KUKA KRL program: f1_Kuka_APT211T03S11.SRC

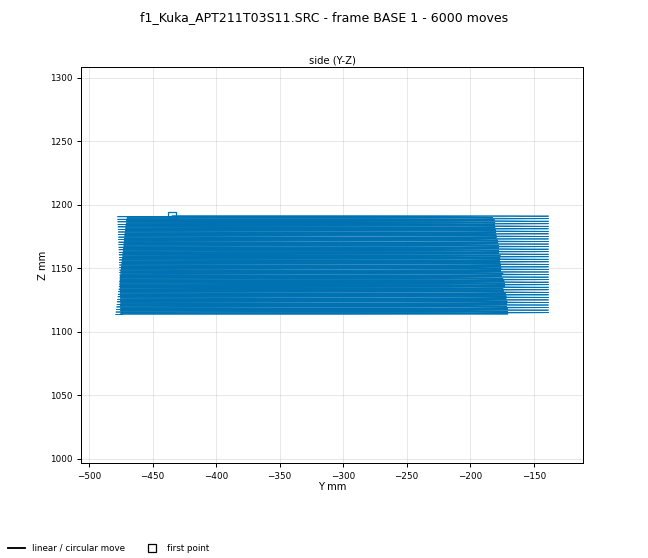
[picture p0: tool path of f1_Kuka_APT211T03S11.SRC in frame BASE 1, 6000 of 6001 moves have a stored position in this frame; points joined in program order, loops and branches not executed]
&ACCESS RVP
&REL 2
&PARAM TEMPLATE = C:\KRC\Roboter\Template\vorgabe
&PARAM EDITMASK = *
DEF f1_Kuka_APT211T03S11()


;FOLD INI;%{PE}%V3.2.0,%MKUKATPBASIS,%CINIT,%VCOMMON,%P
  ;FOLD BAS INI;%{E}%V3.2.0,%MKUKATPBASIS,%CINIT,%VINIT,%P
    GLOBAL INTERRUPT DECL 3 WHEN $STOPMESS==TRUE DO IR_STOPM ( )
    INTERRUPT ON 3
    BAS (#INITMOV,0 )
  ;ENDFOLD (BAS INI)
  ;FOLD USER INI;%{E}%V3.2.0,%MKUKATPUSER,%CINIT,%VINIT,%P
    ;Make your modifications here
  ;ENDFOLD (USER INI)
;ENDFOLD (INI)


;*** Make Null PTP Move
  PTP $pos_act

;*** Auto Load The Correct TOOL Data
  $tool=tool_data[3]

;*** Auto Load The Correct BASE Data
  $base=base_data[1]

  $ADVANCE = 5

;*** Restate Last Velocity
MMPM(30000.0)
SetRPM(6000)
LIN {X -0.088,Y -434.783,Z 1191.509,A 0.000,B 0.000,C 90.000,E1 271.661} C_DIS
LIN {X 0.189,Y -427.658,Z 1191.507,A 0.000,B 0.000,C 90.000,E1 271.318} C_DIS
LIN {X 0.032,Y -420.756,Z 1191.506,A 0.000,B 0.000,C 90.000,E1 271.088} C_DIS
LIN {X -0.167,Y -410.743,Z 1191.504,A 0.000,B 0.000,C 90.000,E1 270.802} C_DIS
LIN {X 0.135,Y -403.684,Z 1191.503,A 0.000,B 0.000,C 90.000,E1 270.573} C_DIS
LIN {X 0.127,Y -392.814,Z 1191.502,A 0.000,B 0.000,C 90.000,E1 270.344} C_DIS
LIN {X 0.051,Y -385.052,Z 1191.501,A 0.000,B 0.000,C 90.000,E1 270.229} C_DIS
LIN {X 0.126,Y -375.484,Z 1191.501,A 0.000,B 0.000,C 90.000,E1 270.115} C_DIS
LIN {X -0.096,Y -368.887,Z 1191.501,A 0.000,B 0.000,C 90.000,E1 270.115} C_DIS
LIN {X -0.083,Y -181.572,Z 1191.500,A 0.000,B 0.000,C 90.000,E1 270.115} C_DIS
LIN {X 0.017,Y -180.908,Z 1191.475,A 0.000,B 0.000,C 90.000,E1 265.527} C_DIS
LIN {X 0.075,Y -180.763,Z 1191.470,A 0.000,B 0.000,C 90.000,E1 264.666} C_DIS
LIN {X -0.034,Y -178.857,Z 1191.442,A 0.000,B 0.000,C 90.000,E1 259.634} C_DIS
LIN {X 0.037,Y -175.900,Z 1191.414,A 0.000,B 0.000,C 90.000,E1 254.519} C_DIS
LIN {X -0.024,Y -174.579,Z 1191.405,A 0.000,B 0.000,C 90.000,E1 252.834} C_DIS
LIN {X 0.011,Y -171.562,Z 1191.381,A 0.000,B 0.000,C 90.000,E1 248.539} C_DIS
LIN {X -0.006,Y -167.786,Z 1191.357,A 0.000,B 0.000,C 90.000,E1 244.229} C_DIS
LIN {X 0.008,Y -166.499,Z 1191.347,A 0.000,B 0.000,C 90.000,E1 242.487} C_DIS
LIN {X 0.004,Y -163.209,Z 1191.328,A 0.000,B 0.000,C 90.000,E1 238.997} C_DIS
LIN {X -0.032,Y -161.174,Z 1191.313,A 0.000,B 0.000,C 90.000,E1 236.373} C_DIS
LIN {X 0.093,Y -157.187,Z 1191.289,A 0.000,B 0.000,C 90.000,E1 231.904} C_DIS
LIN {X 0.015,Y -155.917,Z 1191.279,A 0.000,B 0.000,C 90.000,E1 230.150} C_DIS
LIN {X 0.071,Y -152.169,Z 1191.254,A 0.000,B 0.000,C 90.000,E1 225.648} C_DIS
LIN {X -0.020,Y -150.416,Z 1191.239,A 0.000,B 0.000,C 90.000,E1 222.975} C_DIS
LIN {X -0.094,Y -147.145,Z 1191.214,A 0.000,B 0.000,C 90.000,E1 218.463} C_DIS
LIN {X 0.019,Y -145.703,Z 1191.198,A 0.000,B 0.000,C 90.000,E1 215.678} C_DIS
LIN {X 0.027,Y -143.087,Z 1191.173,A 0.000,B 0.000,C 90.000,E1 211.082} C_DIS
LIN {X 0.032,Y -141.703,Z 1191.152,A 0.000,B 0.000,C 90.000,E1 207.385} C_DIS
LIN {X -0.046,Y -139.468,Z 1191.116,A 0.000,B 0.000,C 90.000,E1 200.918} C_DIS
LIN {X 0.008,Y -139.201,Z 1191.106,A 0.000,B 0.000,C 90.000,E1 199.033} C_DIS
LIN {X 0.071,Y -138.327,Z 1191.054,A 0.000,B 0.000,C 90.000,E1 189.670} C_DIS
LIN {X -0.062,Y -139.443,Z 1191.007,A 0.000,B 0.000,C 90.000,E1 181.318} C_DIS
LIN {X 0.017,Y -140.980,Z 1190.976,A 0.000,B 0.000,C 90.000,E1 175.698} C_DIS
LIN {X -0.033,Y -142.736,Z 1190.956,A 0.000,B 0.000,C 90.000,E1 172.008} C_DIS
LIN {X 0.066,Y -145.126,Z 1190.930,A 0.000,B 0.000,C 90.000,E1 167.353} C_DIS
LIN {X 0.059,Y -147.749,Z 1190.910,A 0.000,B 0.000,C 90.000,E1 163.685} C_DIS
LIN {X -0.001,Y -150.418,Z 1190.889,A 0.000,B 0.000,C 90.000,E1 160.061} C_DIS
LIN {X 0.014,Y -153.858,Z 1190.869,A 0.000,B 0.000,C 90.000,E1 156.433} C_DIS
LIN {X -0.069,Y -157.269,Z 1190.849,A 0.000,B 0.000,C 90.000,E1 152.871} C_DIS
LIN {X 0.008,Y -161.446,Z 1190.829,A 0.000,B 0.000,C 90.000,E1 149.282} C_DIS
LIN {X 0.016,Y -165.646,Z 1190.810,A 0.000,B 0.000,C 90.000,E1 145.754} C_DIS
LIN {X -0.002,Y -170.580,Z 1190.790,A 0.000,B 0.000,C 90.000,E1 142.271} C_DIS
LIN {X -0.095,Y -175.457,Z 1190.771,A 0.000,B 0.000,C 90.000,E1 138.852} C_DIS
LIN {X 0.020,Y -181.080,Z 1190.752,A 0.000,B 0.000,C 90.000,E1 135.405} C_DIS
LIN {X 0.010,Y -186.520,Z 1190.734,A 0.000,B 0.000,C 90.000,E1 132.043} C_DIS
LIN {X -0.048,Y -191.139,Z 1190.720,A 0.000,B 0.000,C 90.000,E1 129.564} C_DIS
LIN {X 0.030,Y -196.938,Z 1190.701,A 0.000,B 0.000,C 90.000,E1 126.251} C_DIS
LIN {X -0.015,Y -201.163,Z 1190.690,A 0.000,B 0.000,C 90.000,E1 124.119} C_DIS
LIN {X 0.133,Y -201.443,Z 1190.689,A 0.000,B 0.000,C 90.000,E1 123.913} C_DIS
LIN {X 0.171,Y -311.509,Z 1190.689,A 0.000,B 0.000,C 90.000,E1 123.913} C_DIS
LIN {X -0.067,Y -315.813,Z 1190.688,A 0.000,B 0.000,C 90.000,E1 123.833} C_DIS
LIN {X 0.069,Y -318.680,Z 1190.687,A 0.000,B 0.000,C 90.000,E1 123.627} C_DIS
LIN {X 0.063,Y -322.419,Z 1190.685,A 0.000,B 0.000,C 90.000,E1 123.245} C_DIS
LIN {X 0.082,Y -325.877,Z 1190.682,A 0.000,B 0.000,C 90.000,E1 122.673} C_DIS
LIN {X -0.013,Y -328.378,Z 1190.678,A 0.000,B 0.000,C 90.000,E1 122.054} C_DIS
LIN {X 0.171,Y -339.358,Z 1190.662,A 0.000,B 0.000,C 90.000,E1 119.205} C_DIS
LIN {X -0.121,Y -351.728,Z 1190.647,A 0.000,B 0.000,C 90.000,E1 116.488} C_DIS
LIN {X -0.053,Y -365.589,Z 1190.632,A 0.000,B 0.000,C 90.000,E1 113.770} C_DIS
LIN {X 0.003,Y -379.265,Z 1190.619,A 0.000,B 0.000,C 90.000,E1 111.408} C_DIS
LIN {X 0.128,Y -394.313,Z 1190.606,A 0.000,B 0.000,C 90.000,E1 109.087} C_DIS
LIN {X -0.003,Y -410.841,Z 1190.594,A 0.000,B 0.000,C 90.000,E1 106.858} C_DIS
LIN {X 0.038,Y -428.965,Z 1190.582,A 0.000,B 0.000,C 90.000,E1 104.662} C_DIS
LIN {X 0.172,Y -448.597,Z 1190.570,A 0.000,B 0.000,C 90.000,E1 102.535} C_DIS
LIN {X 0.088,Y -471.379,Z 1190.558,A 0.000,B 0.000,C 90.000,E1 100.366} C_DIS
LIN {X -0.023,Y -473.312,Z 1190.556,A 0.000,B 0.000,C 90.000,E1 100.141} C_DIS
LIN {X -0.052,Y -474.780,Z 1190.555,A 0.000,B 0.000,C 90.000,E1 99.905} C_DIS
LIN {X 0.143,Y -476.796,Z 1190.552,A 0.000,B 0.000,C 90.000,E1 99.378} C_DIS
LIN {X -0.202,Y -477.678,Z 1190.549,A 0.000,B 0.000,C 90.000,E1 98.916} C_DIS
LIN {X -0.062,Y -477.576,Z 1190.547,A 0.000,B 0.000,C 90.000,E1 98.398} C_DIS
LIN {X 0.151,Y -476.484,Z 1190.544,A 0.000,B 0.000,C 90.000,E1 97.871} C_DIS
LIN {X -0.044,Y -475.517,Z 1190.542,A 0.000,B 0.000,C 90.000,E1 97.644} C_DIS
LIN {X -0.176,Y -474.208,Z 1190.541,A 0.000,B 0.000,C 90.000,E1 97.409} C_DIS
LIN {X -0.051,Y -461.532,Z 1190.531,A 0.000,B 0.000,C 90.000,E1 95.625} C_DIS
LIN {X -0.170,Y -448.957,Z 1190.521,A 0.000,B 0.000,C 90.000,E1 93.841} C_DIS
LIN {X 0.191,Y -433.692,Z 1190.508,A 0.000,B 0.000,C 90.000,E1 91.432} C_DIS
LIN {X 0.019,Y -421.108,Z 1190.496,A 0.000,B 0.000,C 90.000,E1 89.312} C_DIS
LIN {X -0.088,Y -410.843,Z 1190.486,A 0.000,B 0.000,C 90.000,E1 87.421} C_DIS
LIN {X 0.017,Y -400.562,Z 1190.475,A 0.000,B 0.000,C 90.000,E1 85.469} C_DIS
LIN {X -0.061,Y -390.360,Z 1190.464,A 0.000,B 0.000,C 90.000,E1 83.514} C_DIS
LIN {X 0.119,Y -380.156,Z 1190.453,A 0.000,B 0.000,C 90.000,E1 81.489} C_DIS
LIN {X 0.144,Y -371.127,Z 1190.443,A 0.000,B 0.000,C 90.000,E1 79.746} C_DIS
LIN {X 0.074,Y -361.815,Z 1190.433,A 0.000,B 0.000,C 90.000,E1 77.993} C_DIS
LIN {X -0.083,Y -352.243,Z 1190.423,A 0.000,B 0.000,C 90.000,E1 76.228} C_DIS
LIN {X -0.072,Y -340.984,Z 1190.412,A 0.000,B 0.000,C 90.000,E1 74.102} C_DIS
LIN {X -0.123,Y -329.798,Z 1190.400,A 0.000,B 0.000,C 90.000,E1 71.945} C_DIS
LIN {X -0.013,Y -315.928,Z 1190.384,A 0.000,B 0.000,C 90.000,E1 69.082} C_DIS
LIN {X 0.125,Y -300.034,Z 1190.364,A 0.000,B 0.000,C 90.000,E1 65.485} C_DIS
LIN {X 0.133,Y -287.965,Z 1190.347,A 0.000,B 0.000,C 90.000,E1 62.487} C_DIS
LIN {X -0.085,Y -275.372,Z 1190.328,A 0.000,B 0.000,C 90.000,E1 59.125} C_DIS
LIN {X 0.118,Y -263.526,Z 1190.309,A 0.000,B 0.000,C 90.000,E1 55.595} C_DIS
LIN {X 0.082,Y -253.445,Z 1190.291,A 0.000,B 0.000,C 90.000,E1 52.396} C_DIS
LIN {X 0.059,Y -243.968,Z 1190.273,A 0.000,B 0.000,C 90.000,E1 49.138} C_DIS
LIN {X -0.126,Y -234.043,Z 1190.253,A 0.000,B 0.000,C 90.000,E1 45.486} C_DIS
LIN {X 0.035,Y -224.894,Z 1190.232,A 0.000,B 0.000,C 90.000,E1 41.676} C_DIS
LIN {X -0.024,Y -218.244,Z 1190.215,A 0.000,B 0.000,C 90.000,E1 38.624} C_DIS
LIN {X -0.056,Y -210.782,Z 1190.193,A 0.000,B 0.000,C 90.000,E1 34.739} C_DIS
LIN {X -0.101,Y -204.190,Z 1190.171,A 0.000,B 0.000,C 90.000,E1 30.797} C_DIS
LIN {X 0.043,Y -198.271,Z 1190.149,A 0.000,B 0.000,C 90.000,E1 26.744} C_DIS
LIN {X -0.001,Y -193.148,Z 1190.126,A 0.000,B 0.000,C 90.000,E1 22.695} C_DIS
LIN {X -0.037,Y -188.788,Z 1190.103,A 0.000,B 0.000,C 90.000,E1 18.598} C_DIS
LIN {X 0.048,Y -185.390,Z 1190.080,A 0.000,B 0.000,C 90.000,E1 14.426} C_DIS
LIN {X 0.061,Y -182.321,Z 1190.048,A 0.000,B 0.000,C 90.000,E1 8.568} C_DIS
LIN {X 0.047,Y -183.292,Z 1189.965,A 0.000,B 0.000,C 90.000,E1 353.628} C_DIS
LIN {X -0.041,Y -186.535,Z 1189.937,A 0.000,B 0.000,C 90.000,E1 348.634} C_DIS
LIN {X 0.062,Y -190.300,Z 1189.914,A 0.000,B 0.000,C 90.000,E1 344.448} C_DIS
LIN {X -0.067,Y -194.984,Z 1189.891,A 0.000,B 0.000,C 90.000,E1 340.369} C_DIS
LIN {X -0.018,Y -200.311,Z 1189.868,A 0.000,B 0.000,C 90.000,E1 336.282} C_DIS
LIN {X 0.077,Y -206.276,Z 1189.846,A 0.000,B 0.000,C 90.000,E1 332.231} C_DIS
LIN {X 0.003,Y -212.819,Z 1189.824,A 0.000,B 0.000,C 90.000,E1 328.280} C_DIS
LIN {X 0.040,Y -219.997,Z 1189.802,A 0.000,B 0.000,C 90.000,E1 324.356} C_DIS
LIN {X 0.105,Y -226.235,Z 1189.785,A 0.000,B 0.000,C 90.000,E1 321.251} C_DIS
LIN {X -0.055,Y -233.325,Z 1189.768,A 0.000,B 0.000,C 90.000,E1 318.243} C_DIS
LIN {X 0.088,Y -242.603,Z 1189.749,A 0.000,B 0.000,C 90.000,E1 314.838} C_DIS
LIN {X 0.016,Y -253.506,Z 1189.731,A 0.000,B 0.000,C 90.000,E1 311.553} C_DIS
LIN {X -0.049,Y -265.573,Z 1189.713,A 0.000,B 0.000,C 90.000,E1 308.338} C_DIS
LIN {X -0.082,Y -275.913,Z 1189.699,A 0.000,B 0.000,C 90.000,E1 305.884} C_DIS
LIN {X 0.028,Y -287.499,Z 1189.686,A 0.000,B 0.000,C 90.000,E1 303.452} C_DIS
LIN {X 0.087,Y -298.373,Z 1189.675,A 0.000,B 0.000,C 90.000,E1 301.416} C_DIS
LIN {X -0.029,Y -312.380,Z 1189.662,A 0.000,B 0.000,C 90.000,E1 299.127} C_DIS
LIN {X 0.042,Y -325.764,Z 1189.651,A 0.000,B 0.000,C 90.000,E1 297.180} C_DIS
LIN {X 0.033,Y -333.126,Z 1189.646,A 0.000,B 0.000,C 90.000,E1 296.232} C_DIS
LIN {X -0.148,Y -354.255,Z 1189.632,A 0.000,B 0.000,C 90.000,E1 293.823} C_DIS
LIN {X 0.035,Y -378.498,Z 1189.618,A 0.000,B 0.000,C 90.000,E1 291.280} C_DIS
LIN {X -0.113,Y -394.625,Z 1189.610,A 0.000,B 0.000,C 90.000,E1 289.758} C_DIS
LIN {X -0.054,Y -407.817,Z 1189.603,A 0.000,B 0.000,C 90.000,E1 288.471} C_DIS
LIN {X -0.106,Y -417.892,Z 1189.597,A 0.000,B 0.000,C 90.000,E1 287.457} C_DIS
LIN {X 0.013,Y -427.679,Z 1189.591,A 0.000,B 0.000,C 90.000,E1 286.386} C_DIS
LIN {X -0.205,Y -434.725,Z 1189.587,A 0.000,B 0.000,C 90.000,E1 285.607} C_DIS
LIN {X 0.060,Y -441.189,Z 1189.582,A 0.000,B 0.000,C 90.000,E1 284.773} C_DIS
LIN {X -0.160,Y -446.904,Z 1189.578,A 0.000,B 0.000,C 90.000,E1 284.008} C_DIS
LIN {X 0.220,Y -451.991,Z 1189.573,A 0.000,B 0.000,C 90.000,E1 283.175} C_DIS
LIN {X 0.095,Y -456.430,Z 1189.569,A 0.000,B 0.000,C 90.000,E1 282.411} C_DIS
LIN {X -0.083,Y -460.057,Z 1189.565,A 0.000,B 0.000,C 90.000,E1 281.658} C_DIS
LIN {X -0.138,Y -463.096,Z 1189.560,A 0.000,B 0.000,C 90.000,E1 280.894} C_DIS
LIN {X -0.015,Y -464.741,Z 1189.558,A 0.000,B 0.000,C 90.000,E1 280.366} C_DIS
LIN {X 0.181,Y -467.347,Z 1189.552,A 0.000,B 0.000,C 90.000,E1 279.321} C_DIS
LIN {X -0.207,Y -468.452,Z 1189.549,A 0.000,B 0.000,C 90.000,E1 278.859} C_DIS
LIN {X -0.123,Y -469.349,Z 1189.546,A 0.000,B 0.000,C 90.000,E1 278.341} C_DIS
LIN {X 0.035,Y -470.033,Z 1189.543,A 0.000,B 0.000,C 90.000,E1 277.814} C_DIS
LIN {X 0.132,Y -470.374,Z 1189.541,A 0.000,B 0.000,C 90.000,E1 277.296} C_DIS
LIN {X 0.234,Y -470.270,Z 1189.538,A 0.000,B 0.000,C 90.000,E1 276.777} C_DIS
LIN {X -0.128,Y -469.820,Z 1189.535,A 0.000,B 0.000,C 90.000,E1 276.315} C_DIS
LIN {X -0.025,Y -468.861,Z 1189.532,A 0.000,B 0.000,C 90.000,E1 275.796} C_DIS
LIN {X 0.075,Y -467.463,Z 1189.529,A 0.000,B 0.000,C 90.000,E1 275.277} C_DIS
LIN {X 0.167,Y -465.601,Z 1189.527,A 0.000,B 0.000,C 90.000,E1 274.759} C_DIS
LIN {X 0.214,Y -463.174,Z 1189.524,A 0.000,B 0.000,C 90.000,E1 274.245} C_DIS
LIN {X -0.181,Y -460.133,Z 1189.521,A 0.000,B 0.000,C 90.000,E1 273.784} C_DIS
LIN {X 0.058,Y -458.329,Z 1189.520,A 0.000,B 0.000,C 90.000,E1 273.498} C_DIS
LIN {X 0.094,Y -453.949,Z 1189.517,A 0.000,B 0.000,C 90.000,E1 272.980} C_DIS
LIN {X -0.130,Y -451.317,Z 1189.515,A 0.000,B 0.000,C 90.000,E1 272.751} C_DIS
LIN {X 0.173,Y -448.439,Z 1189.514,A 0.000,B 0.000,C 90.000,E1 272.465} C_DIS
LIN {X 0.188,Y -442.175,Z 1189.511,A 0.000,B 0.000,C 90.000,E1 272.007} C_DIS
LIN {X -0.055,Y -435.315,Z 1189.509,A 0.000,B 0.000,C 90.000,E1 271.661} C_DIS
LIN {X 0.207,Y -428.243,Z 1189.507,A 0.000,B 0.000,C 90.000,E1 271.318} C_DIS
LIN {X 0.011,Y -421.326,Z 1189.506,A 0.000,B 0.000,C 90.000,E1 271.088} C_DIS
LIN {X 0.195,Y -411.152,Z 1189.504,A 0.000,B 0.000,C 90.000,E1 270.745} C_DIS
LIN {X 0.107,Y -404.249,Z 1189.503,A 0.000,B 0.000,C 90.000,E1 270.573} C_DIS
LIN {X 0.099,Y -393.448,Z 1189.502,A 0.000,B 0.000,C 90.000,E1 270.344} C_DIS
LIN {X 0.008,Y -385.768,Z 1189.501,A 0.000,B 0.000,C 90.000,E1 270.229} C_DIS
LIN {X 0.067,Y -376.435,Z 1189.501,A 0.000,B 0.000,C 90.000,E1 270.115} C_DIS
LIN {X 0.134,Y -365.555,Z 1189.500,A 0.000,B 0.000,C 90.000,E1 270.057} C_DIS
LIN {X 0.046,Y -181.570,Z 1189.500,A 0.000,B 0.000,C 90.000,E1 270.057} C_DIS
LIN {X 0.067,Y -180.855,Z 1189.472,A 0.000,B 0.000,C 90.000,E1 264.951} C_DIS
LIN {X -0.058,Y -178.967,Z 1189.444,A 0.000,B 0.000,C 90.000,E1 259.926} C_DIS
LIN {X -0.047,Y -177.920,Z 1189.435,A 0.000,B 0.000,C 90.000,E1 258.229} C_DIS
LIN {X -0.032,Y -175.556,Z 1189.411,A 0.000,B 0.000,C 90.000,E1 253.976} C_DIS
LIN {X -0.026,Y -172.287,Z 1189.387,A 0.000,B 0.000,C 90.000,E1 249.699} C_DIS
LIN {X -0.048,Y -171.765,Z 1189.382,A 0.000,B 0.000,C 90.000,E1 248.847} C_DIS
LIN {X 0.030,Y -167.366,Z 1189.354,A 0.000,B 0.000,C 90.000,E1 243.640} C_DIS
LIN {X -0.036,Y -166.756,Z 1189.349,A 0.000,B 0.000,C 90.000,E1 242.794} C_DIS
LIN {X 0.024,Y -162.735,Z 1189.325,A 0.000,B 0.000,C 90.000,E1 238.408} C_DIS
LIN {X 0.085,Y -161.426,Z 1189.315,A 0.000,B 0.000,C 90.000,E1 236.628} C_DIS
LIN {X -0.095,Y -157.419,Z 1189.290,A 0.000,B 0.000,C 90.000,E1 232.271} C_DIS
LIN {X 0.059,Y -155.422,Z 1189.275,A 0.000,B 0.000,C 90.000,E1 229.542} C_DIS
LIN {X -0.010,Y -151.747,Z 1189.250,A 0.000,B 0.000,C 90.000,E1 225.081} C_DIS
LIN {X 0.000,Y -149.946,Z 1189.235,A 0.000,B 0.000,C 90.000,E1 222.366} C_DIS
LIN {X 0.028,Y -146.791,Z 1189.210,A 0.000,B 0.000,C 90.000,E1 217.810} C_DIS
LIN {X -0.071,Y -145.365,Z 1189.195,A 0.000,B 0.000,C 90.000,E1 215.105} C_DIS
LIN {X 0.045,Y -142.431,Z 1189.164,A 0.000,B 0.000,C 90.000,E1 209.539} C_DIS
LIN {X -0.031,Y -141.421,Z 1189.149,A 0.000,B 0.000,C 90.000,E1 206.796} C_DIS
LIN {X -0.049,Y -139.362,Z 1189.113,A 0.000,B 0.000,C 90.000,E1 200.301} C_DIS
LIN {X 0.069,Y -138.805,Z 1189.097,A 0.000,B 0.000,C 90.000,E1 197.457} C_DIS
LIN {X -0.012,Y -138.350,Z 1189.056,A 0.000,B 0.000,C 90.000,E1 190.018} C_DIS
LIN {X -0.036,Y -139.544,Z 1189.004,A 0.000,B 0.000,C 90.000,E1 180.688} C_DIS
LIN {X 0.056,Y -141.245,Z 1188.973,A 0.000,B 0.000,C 90.000,E1 175.065} C_DIS
LIN {X 0.015,Y -142.614,Z 1188.957,A 0.000,B 0.000,C 90.000,E1 172.299} C_DIS
LIN {X -0.033,Y -144.930,Z 1188.932,A 0.000,B 0.000,C 90.000,E1 167.701} C_DIS
LIN {X -0.040,Y -147.559,Z 1188.911,A 0.000,B 0.000,C 90.000,E1 164.031} C_DIS
LIN {X -0.009,Y -150.165,Z 1188.891,A 0.000,B 0.000,C 90.000,E1 160.369} C_DIS
LIN {X 0.000,Y -153.538,Z 1188.871,A 0.000,B 0.000,C 90.000,E1 156.741} C_DIS
LIN {X 0.052,Y -156.956,Z 1188.851,A 0.000,B 0.000,C 90.000,E1 153.127} C_DIS
LIN {X -0.012,Y -161.062,Z 1188.831,A 0.000,B 0.000,C 90.000,E1 149.587} C_DIS
LIN {X 0.072,Y -163.170,Z 1188.821,A 0.000,B 0.000,C 90.000,E1 147.788} C_DIS
LIN {X -0.056,Y -167.590,Z 1188.802,A 0.000,B 0.000,C 90.000,E1 144.322} C_DIS
LIN {X -0.011,Y -171.419,Z 1188.787,A 0.000,B 0.000,C 90.000,E1 141.698} C_DIS
LIN {X 0.027,Y -176.336,Z 1188.768,A 0.000,B 0.000,C 90.000,E1 138.243} C_DIS
LIN {X -0.105,Y -180.626,Z 1188.754,A 0.000,B 0.000,C 90.000,E1 135.729} C_DIS
LIN {X 0.010,Y -186.027,Z 1188.735,A 0.000,B 0.000,C 90.000,E1 132.324} C_DIS
LIN {X 0.072,Y -190.663,Z 1188.721,A 0.000,B 0.000,C 90.000,E1 129.806} C_DIS
LIN {X 0.106,Y -196.414,Z 1188.703,A 0.000,B 0.000,C 90.000,E1 126.503} C_DIS
LIN {X -0.033,Y -201.388,Z 1188.689,A 0.000,B 0.000,C 90.000,E1 123.992} C_DIS
LIN {X -0.102,Y -311.074,Z 1188.689,A 0.000,B 0.000,C 90.000,E1 123.992} C_DIS
LIN {X -0.153,Y -312.007,Z 1188.689,A 0.000,B 0.000,C 90.000,E1 123.992} C_DIS
LIN {X 0.048,Y -316.708,Z 1188.688,A 0.000,B 0.000,C 90.000,E1 123.785} C_DIS
LIN {X -0.013,Y -319.086,Z 1188.687,A 0.000,B 0.000,C 90.000,E1 123.627} C_DIS
LIN {X -0.047,Y -322.298,Z 1188.685,A 0.000,B 0.000,C 90.000,E1 123.293} C_DIS
LIN {X -0.078,Y -324.275,Z 1188.683,A 0.000,B 0.000,C 90.000,E1 123.007} C_DIS
LIN {X -0.012,Y -325.822,Z 1188.682,A 0.000,B 0.000,C 90.000,E1 122.704} C_DIS
LIN {X -0.093,Y -328.297,Z 1188.678,A 0.000,B 0.000,C 90.000,E1 122.084} C_DIS
LIN {X -0.195,Y -339.269,Z 1188.662,A 0.000,B 0.000,C 90.000,E1 119.283} C_DIS
LIN {X -0.024,Y -351.630,Z 1188.647,A 0.000,B 0.000,C 90.000,E1 116.488} C_DIS
LIN {X 0.045,Y -365.482,Z 1188.632,A 0.000,B 0.000,C 90.000,E1 113.770} C_DIS
LIN {X 0.101,Y -379.149,Z 1188.619,A 0.000,B 0.000,C 90.000,E1 111.408} C_DIS
LIN {X -0.145,Y -394.188,Z 1188.606,A 0.000,B 0.000,C 90.000,E1 109.141} C_DIS
LIN {X 0.098,Y -410.706,Z 1188.594,A 0.000,B 0.000,C 90.000,E1 106.858} C_DIS
LIN {X 0.139,Y -428.819,Z 1188.582,A 0.000,B 0.000,C 90.000,E1 104.662} C_DIS
LIN {X -0.166,Y -448.444,Z 1188.570,A 0.000,B 0.000,C 90.000,E1 102.591} C_DIS
LIN {X 0.182,Y -471.233,Z 1188.558,A 0.000,B 0.000,C 90.000,E1 100.366} C_DIS
LIN {X 0.075,Y -473.176,Z 1188.556,A 0.000,B 0.000,C 90.000,E1 100.141} C_DIS
LIN {X 0.052,Y -474.653,Z 1188.555,A 0.000,B 0.000,C 90.000,E1 99.905} C_DIS
LIN {X -0.085,Y -475.831,Z 1188.554,A 0.000,B 0.000,C 90.000,E1 99.670} C_DIS
LIN {X 0.247,Y -476.688,Z 1188.552,A 0.000,B 0.000,C 90.000,E1 99.378} C_DIS
LIN {X -0.093,Y -477.583,Z 1188.549,A 0.000,B 0.000,C 90.000,E1 98.916} C_DIS
LIN {X 0.047,Y -477.498,Z 1188.547,A 0.000,B 0.000,C 90.000,E1 98.398} C_DIS
LIN {X 0.259,Y -476.423,Z 1188.544,A 0.000,B 0.000,C 90.000,E1 97.871} C_DIS
LIN {X 0.063,Y -475.465,Z 1188.542,A 0.000,B 0.000,C 90.000,E1 97.644} C_DIS
LIN {X -0.068,Y -474.169,Z 1188.541,A 0.000,B 0.000,C 90.000,E1 97.409} C_DIS
LIN {X 0.053,Y -461.526,Z 1188.531,A 0.000,B 0.000,C 90.000,E1 95.625} C_DIS
LIN {X -0.069,Y -448.940,Z 1188.521,A 0.000,B 0.000,C 90.000,E1 93.841} C_DIS
LIN {X 0.015,Y -432.023,Z 1188.507,A 0.000,B 0.000,C 90.000,E1 91.203} C_DIS
LIN {X -0.190,Y -419.594,Z 1188.495,A 0.000,B 0.000,C 90.000,E1 89.083} C_DIS
LIN {X 0.081,Y -409.356,Z 1188.484,A 0.000,B 0.000,C 90.000,E1 87.135} C_DIS
LIN {X -0.175,Y -397.580,Z 1188.472,A 0.000,B 0.000,C 90.000,E1 84.951} C_DIS
LIN {X 0.116,Y -385.933,Z 1188.459,A 0.000,B 0.000,C 90.000,E1 82.648} C_DIS
LIN {X -0.188,Y -377.121,Z 1188.450,A 0.000,B 0.000,C 90.000,E1 80.971} C_DIS
LIN {X -0.147,Y -367.992,Z 1188.440,A 0.000,B 0.000,C 90.000,E1 79.218} C_DIS
LIN {X 0.086,Y -358.579,Z 1188.430,A 0.000,B 0.000,C 90.000,E1 77.409} C_DIS
LIN {X -0.131,Y -348.939,Z 1188.420,A 0.000,B 0.000,C 90.000,E1 75.644} C_DIS
LIN {X -0.102,Y -337.694,Z 1188.408,A 0.000,B 0.000,C 90.000,E1 73.504} C_DIS
LIN {X 0.157,Y -325.032,Z 1188.394,A 0.000,B 0.000,C 90.000,E1 70.967} C_DIS
LIN {X 0.050,Y -309.920,Z 1188.377,A 0.000,B 0.000,C 90.000,E1 67.794} C_DIS
LIN {X -0.043,Y -294.519,Z 1188.357,A 0.000,B 0.000,C 90.000,E1 64.204} C_DIS
LIN {X -0.078,Y -281.468,Z 1188.338,A 0.000,B 0.000,C 90.000,E1 60.845} C_DIS
LIN {X -0.042,Y -270.440,Z 1188.321,A 0.000,B 0.000,C 90.000,E1 57.740} C_DIS
LIN {X 0.022,Y -259.981,Z 1188.303,A 0.000,B 0.000,C 90.000,E1 54.562} C_DIS
LIN {X 0.039,Y -250.047,Z 1188.285,A 0.000,B 0.000,C 90.000,E1 51.331} C_DIS
LIN {X 0.086,Y -241.753,Z 1188.269,A 0.000,B 0.000,C 90.000,E1 48.405} C_DIS
LIN {X -0.017,Y -231.953,Z 1188.248,A 0.000,B 0.000,C 90.000,E1 44.717} C_DIS
LIN {X 0.079,Y -223.002,Z 1188.227,A 0.000,B 0.000,C 90.000,E1 40.906} C_DIS
LIN {X -0.024,Y -214.998,Z 1188.206,A 0.000,B 0.000,C 90.000,E1 37.076} C_DIS
LIN {X -0.059,Y -207.868,Z 1188.184,A 0.000,B 0.000,C 90.000,E1 33.166} C_DIS
LIN {X 0.052,Y -201.531,Z 1188.162,A 0.000,B 0.000,C 90.000,E1 29.155} C_DIS
LIN {X -0.070,Y -195.841,Z 1188.140,A 0.000,B 0.000,C 90.000,E1 25.155} C_DIS
LIN {X 0.019,Y -191.047,Z 1188.117,A 0.000,B 0.000,C 90.000,E1 21.046} C_DIS
LIN {X 0.037,Y -187.008,Z 1188.094,A 0.000,B 0.000,C 90.000,E1 16.913} C_DIS
LIN {X -0.079,Y -183.534,Z 1188.066,A 0.000,B 0.000,C 90.000,E1 11.951} C_DIS
LIN {X -0.038,Y -181.032,Z 1188.029,A 0.000,B 0.000,C 90.000,E1 5.220} C_DIS
LIN {X -0.034,Y -182.540,Z 1187.969,A 0.000,B 0.000,C 90.000,E1 354.489} C_DIS
LIN {X -0.021,Y -185.557,Z 1187.941,A 0.000,B 0.000,C 90.000,E1 349.454} C_DIS
LIN {X 0.005,Y -189.126,Z 1187.918,A 0.000,B 0.000,C 90.000,E1 345.283} C_DIS
LIN {X 0.025,Y -193.650,Z 1187.895,A 0.000,B 0.000,C 90.000,E1 341.148} C_DIS
LIN {X 0.071,Y -198.868,Z 1187.873,A 0.000,B 0.000,C 90.000,E1 337.050} C_DIS
LIN {X -0.064,Y -204.695,Z 1187.850,A 0.000,B 0.000,C 90.000,E1 333.050} C_DIS
LIN {X -0.105,Y -211.122,Z 1187.828,A 0.000,B 0.000,C 90.000,E1 329.076} C_DIS
LIN {X 0.069,Y -216.773,Z 1187.811,A 0.000,B 0.000,C 90.000,E1 325.881} C_DIS
LIN {X -0.046,Y -224.311,Z 1187.789,A 0.000,B 0.000,C 90.000,E1 322.029} C_DIS
LIN {X 0.099,Y -231.243,Z 1187.772,A 0.000,B 0.000,C 90.000,E1 318.933} C_DIS
LIN {X -0.123,Y -239.232,Z 1187.755,A 0.000,B 0.000,C 90.000,E1 315.972} C_DIS
LIN {X 0.055,Y -247.191,Z 1187.741,A 0.000,B 0.000,C 90.000,E1 313.338} C_DIS
LIN {X -0.058,Y -258.672,Z 1187.723,A 0.000,B 0.000,C 90.000,E1 310.092} C_DIS
LIN {X 0.062,Y -271.331,Z 1187.705,A 0.000,B 0.000,C 90.000,E1 306.870} C_DIS
LIN {X -0.112,Y -280.752,Z 1187.693,A 0.000,B 0.000,C 90.000,E1 304.818} C_DIS
LIN {X -0.071,Y -294.707,Z 1187.678,A 0.000,B 0.000,C 90.000,E1 302.084} C_DIS
LIN {X 0.032,Y -310.433,Z 1187.663,A 0.000,B 0.000,C 90.000,E1 299.411} C_DIS
LIN {X 0.075,Y -323.549,Z 1187.653,A 0.000,B 0.000,C 90.000,E1 297.462} C_DIS
LIN {X -0.150,Y -333.237,Z 1187.646,A 0.000,B 0.000,C 90.000,E1 296.232} C_DIS
LIN {X -0.066,Y -354.420,Z 1187.632,A 0.000,B 0.000,C 90.000,E1 293.770} C_DIS
LIN {X 0.102,Y -381.390,Z 1187.617,A 0.000,B 0.000,C 90.000,E1 290.972} C_DIS
LIN {X 0.004,Y -394.903,Z 1187.609,A 0.000,B 0.000,C 90.000,E1 289.704} C_DIS
LIN {X 0.131,Y -408.049,Z 1187.602,A 0.000,B 0.000,C 90.000,E1 288.417} C_DIS
LIN {X -0.128,Y -415.597,Z 1187.598,A 0.000,B 0.000,C 90.000,E1 287.692} C_DIS
LIN {X 0.002,Y -425.532,Z 1187.592,A 0.000,B 0.000,C 90.000,E1 286.622} C_DIS
LIN {X -0.225,Y -432.710,Z 1187.588,A 0.000,B 0.000,C 90.000,E1 285.843} C_DIS
LIN {X 0.013,Y -439.396,Z 1187.583,A 0.000,B 0.000,C 90.000,E1 285.009} C_DIS
LIN {X -0.217,Y -445.358,Z 1187.579,A 0.000,B 0.000,C 90.000,E1 284.245} C_DIS
LIN {X 0.142,Y -450.579,Z 1187.575,A 0.000,B 0.000,C 90.000,E1 283.411} C_DIS
LIN {X 0.010,Y -455.248,Z 1187.570,A 0.000,B 0.000,C 90.000,E1 282.647} C_DIS
LIN {X -0.090,Y -459.128,Z 1187.566,A 0.000,B 0.000,C 90.000,E1 281.883} C_DIS
LIN {X -0.077,Y -461.337,Z 1187.563,A 0.000,B 0.000,C 90.000,E1 281.366} C_DIS
LIN {X 0.044,Y -463.279,Z 1187.560,A 0.000,B 0.000,C 90.000,E1 280.838} C_DIS
LIN {X 0.170,Y -464.930,Z 1187.557,A 0.000,B 0.000,C 90.000,E1 280.310} C_DIS
LIN {X -0.091,Y -467.631,Z 1187.552,A 0.000,B 0.000,C 90.000,E1 279.321} C_DIS
LIN {X -0.015,Y -468.781,Z 1187.549,A 0.000,B 0.000,C 90.000,E1 278.803} C_DIS
LIN {X 0.140,Y -469.685,Z 1187.546,A 0.000,B 0.000,C 90.000,E1 278.276} C_DIS
LIN {X 0.233,Y -470.354,Z 1187.543,A 0.000,B 0.000,C 90.000,E1 277.757} C_DIS
LIN {X -0.135,Y -470.647,Z 1187.540,A 0.000,B 0.000,C 90.000,E1 277.296} C_DIS
LIN {X -0.030,Y -470.570,Z 1187.538,A 0.000,B 0.000,C 90.000,E1 276.777} C_DIS
LIN {X 0.076,Y -470.046,Z 1187.535,A 0.000,B 0.000,C 90.000,E1 276.258} C_DIS
LIN {X 0.181,Y -469.022,Z 1187.532,A 0.000,B 0.000,C 90.000,E1 275.739} C_DIS
LIN {X -0.183,Y -467.584,Z 1187.529,A 0.000,B 0.000,C 90.000,E1 275.277} C_DIS
LIN {X -0.089,Y -465.737,Z 1187.526,A 0.000,B 0.000,C 90.000,E1 274.759} C_DIS
LIN {X -0.041,Y -463.296,Z 1187.524,A 0.000,B 0.000,C 90.000,E1 274.245} C_DIS
LIN {X 0.026,Y -460.225,Z 1187.521,A 0.000,B 0.000,C 90.000,E1 273.726} C_DIS
LIN {X 0.048,Y -456.277,Z 1187.518,A 0.000,B 0.000,C 90.000,E1 273.212} C_DIS
LIN {X -0.154,Y -453.941,Z 1187.516,A 0.000,B 0.000,C 90.000,E1 272.980} C_DIS
LIN {X 0.074,Y -451.280,Z 1187.515,A 0.000,B 0.000,C 90.000,E1 272.694} C_DIS
LIN {X -0.189,Y -445.173,Z 1187.512,A 0.000,B 0.000,C 90.000,E1 272.236} C_DIS
LIN {X -0.057,Y -442.036,Z 1187.511,A 0.000,B 0.000,C 90.000,E1 272.007} C_DIS
LIN {X 0.104,Y -435.095,Z 1187.509,A 0.000,B 0.000,C 90.000,E1 271.604} C_DIS
LIN {X -0.058,Y -427.955,Z 1187.507,A 0.000,B 0.000,C 90.000,E1 271.318} C_DIS
LIN {X 0.188,Y -421.041,Z 1187.506,A 0.000,B 0.000,C 90.000,E1 271.031} C_DIS
LIN {X -0.041,Y -410.732,Z 1187.504,A 0.000,B 0.000,C 90.000,E1 270.745} C_DIS
LIN {X 0.135,Y -400.152,Z 1187.503,A 0.000,B 0.000,C 90.000,E1 270.458} C_DIS
LIN {X -0.138,Y -389.157,Z 1187.501,A 0.000,B 0.000,C 90.000,E1 270.286} C_DIS
LIN {X -0.147,Y -380.607,Z 1187.501,A 0.000,B 0.000,C 90.000,E1 270.172} C_DIS
LIN {X 0.157,Y -371.815,Z 1187.500,A 0.000,B 0.000,C 90.000,E1 270.057} C_DIS
LIN {X 0.083,Y -368.300,Z 1187.500,A 0.000,B 0.000,C 90.000,E1 270.057} C_DIS
LIN {X 0.005,Y -181.569,Z 1187.500,A 0.000,B 0.000,C 90.000,E1 270.057} C_DIS
LIN {X -0.074,Y -180.907,Z 1187.475,A 0.000,B 0.000,C 90.000,E1 265.527} C_DIS
LIN {X -0.017,Y -180.751,Z 1187.470,A 0.000,B 0.000,C 90.000,E1 264.666} C_DIS
LIN {X 0.051,Y -178.843,Z 1187.442,A 0.000,B 0.000,C 90.000,E1 259.577} C_DIS
LIN {X -0.053,Y -175.887,Z 1187.414,A 0.000,B 0.000,C 90.000,E1 254.519} C_DIS
LIN {X 0.054,Y -174.554,Z 1187.404,A 0.000,B 0.000,C 90.000,E1 252.779} C_DIS
LIN {X -0.077,Y -171.538,Z 1187.381,A 0.000,B 0.000,C 90.000,E1 248.539} C_DIS
LIN {X -0.021,Y -167.764,Z 1187.357,A 0.000,B 0.000,C 90.000,E1 244.204} C_DIS
LIN {X -0.079,Y -166.470,Z 1187.347,A 0.000,B 0.000,C 90.000,E1 242.487} C_DIS
LIN {X 0.058,Y -163.185,Z 1187.328,A 0.000,B 0.000,C 90.000,E1 238.948} C_DIS
LIN {X -0.027,Y -161.146,Z 1187.313,A 0.000,B 0.000,C 90.000,E1 236.342} C_DIS
LIN {X 0.008,Y -157.164,Z 1187.288,A 0.000,B 0.000,C 90.000,E1 231.904} C_DIS
LIN {X 0.032,Y -155.896,Z 1187.278,A 0.000,B 0.000,C 90.000,E1 230.114} C_DIS
LIN {X -0.011,Y -152.146,Z 1187.254,A 0.000,B 0.000,C 90.000,E1 225.648} C_DIS
LIN {X 0.009,Y -150.395,Z 1187.239,A 0.000,B 0.000,C 90.000,E1 222.933} C_DIS
LIN {X 0.033,Y -147.126,Z 1187.213,A 0.000,B 0.000,C 90.000,E1 218.382} C_DIS
LIN {X 0.024,Y -145.689,Z 1187.198,A 0.000,B 0.000,C 90.000,E1 215.644} C_DIS
LIN {X 0.021,Y -143.071,Z 1187.173,A 0.000,B 0.000,C 90.000,E1 211.052} C_DIS
LIN {X -0.047,Y -141.692,Z 1187.152,A 0.000,B 0.000,C 90.000,E1 207.385} C_DIS
LIN {X 0.007,Y -139.462,Z 1187.116,A 0.000,B 0.000,C 90.000,E1 200.865} C_DIS
LIN {X -0.069,Y -139.195,Z 1187.106,A 0.000,B 0.000,C 90.000,E1 199.033} C_DIS
LIN {X -0.006,Y -138.325,Z 1187.054,A 0.000,B 0.000,C 90.000,E1 189.670} C_DIS
LIN {X -0.001,Y -139.450,Z 1187.007,A 0.000,B 0.000,C 90.000,E1 181.260} C_DIS
LIN {X -0.062,Y -140.994,Z 1186.976,A 0.000,B 0.000,C 90.000,E1 175.698} C_DIS
LIN {X 0.029,Y -142.748,Z 1186.955,A 0.000,B 0.000,C 90.000,E1 171.951} C_DIS
LIN {X -0.015,Y -145.147,Z 1186.930,A 0.000,B 0.000,C 90.000,E1 167.353} C_DIS
LIN {X -0.021,Y -147.770,Z 1186.909,A 0.000,B 0.000,C 90.000,E1 163.685} C_DIS
LIN {X 0.058,Y -150.444,Z 1186.889,A 0.000,B 0.000,C 90.000,E1 160.007} C_DIS
LIN {X -0.007,Y -153.890,Z 1186.869,A 0.000,B 0.000,C 90.000,E1 156.410} C_DIS
LIN {X -0.013,Y -157.300,Z 1186.849,A 0.000,B 0.000,C 90.000,E1 152.820} C_DIS
LIN {X 0.005,Y -161.486,Z 1186.829,A 0.000,B 0.000,C 90.000,E1 149.253} C_DIS
LIN {X 0.021,Y -165.684,Z 1186.810,A 0.000,B 0.000,C 90.000,E1 145.722} C_DIS
LIN {X -0.092,Y -170.626,Z 1186.790,A 0.000,B 0.000,C 90.000,E1 142.271} C_DIS
LIN {X 0.062,Y -175.503,Z 1186.771,A 0.000,B 0.000,C 90.000,E1 138.771} C_DIS
LIN {X -0.072,Y -181.123,Z 1186.752,A 0.000,B 0.000,C 90.000,E1 135.405} C_DIS
LIN {X 0.056,Y -186.571,Z 1186.733,A 0.000,B 0.000,C 90.000,E1 132.000} C_DIS
LIN {X 0.005,Y -191.184,Z 1186.720,A 0.000,B 0.000,C 90.000,E1 129.519} C_DIS
LIN {X 0.051,Y -196.991,Z 1186.701,A 0.000,B 0.000,C 90.000,E1 126.217} C_DIS
LIN {X 0.038,Y -201.139,Z 1186.690,A 0.000,B 0.000,C 90.000,E1 124.119} C_DIS
LIN {X 0.042,Y -201.352,Z 1186.689,A 0.000,B 0.000,C 90.000,E1 123.992} C_DIS
LIN {X 0.028,Y -311.032,Z 1186.689,A 0.000,B 0.000,C 90.000,E1 123.992} C_DIS
LIN {X 0.041,Y -317.019,Z 1186.688,A 0.000,B 0.000,C 90.000,E1 123.785} C_DIS
LIN {X -0.001,Y -319.761,Z 1186.687,A 0.000,B 0.000,C 90.000,E1 123.579} C_DIS
LIN {X 0.190,Y -323.532,Z 1186.684,A 0.000,B 0.000,C 90.000,E1 123.086} C_DIS
LIN {X 0.000,Y -325.355,Z 1186.682,A 0.000,B 0.000,C 90.000,E1 122.801} C_DIS
LIN {X 0.082,Y -326.773,Z 1186.680,A 0.000,B 0.000,C 90.000,E1 122.467} C_DIS
LIN {X 0.064,Y -338.856,Z 1186.663,A 0.000,B 0.000,C 90.000,E1 119.333} C_DIS
LIN {X 0.072,Y -351.166,Z 1186.648,A 0.000,B 0.000,C 90.000,E1 116.565} C_DIS
LIN {X -0.199,Y -364.969,Z 1186.633,A 0.000,B 0.000,C 90.000,E1 113.898} C_DIS
LIN {X -0.163,Y -378.586,Z 1186.620,A 0.000,B 0.000,C 90.000,E1 111.535} C_DIS
LIN {X -0.058,Y -393.571,Z 1186.607,A 0.000,B 0.000,C 90.000,E1 109.214} C_DIS
LIN {X -0.090,Y -410.031,Z 1186.594,A 0.000,B 0.000,C 90.000,E1 106.968} C_DIS
LIN {X -0.084,Y -428.083,Z 1186.582,A 0.000,B 0.000,C 90.000,E1 104.773} C_DIS
LIN {X -0.015,Y -447.677,Z 1186.570,A 0.000,B 0.000,C 90.000,E1 102.647} C_DIS
LIN {X -0.249,Y -470.505,Z 1186.558,A 0.000,B 0.000,C 90.000,E1 100.489} C_DIS
LIN {X -0.216,Y -472.556,Z 1186.557,A 0.000,B 0.000,C 90.000,E1 100.254} C_DIS
LIN {X 0.107,Y -474.241,Z 1186.555,A 0.000,B 0.000,C 90.000,E1 99.962} C_DIS
LIN {X -0.038,Y -475.506,Z 1186.554,A 0.000,B 0.000,C 90.000,E1 99.726} C_DIS
LIN {X 0.085,Y -477.067,Z 1186.551,A 0.000,B 0.000,C 90.000,E1 99.208} C_DIS
LIN {X -0.255,Y -477.576,Z 1186.548,A 0.000,B 0.000,C 90.000,E1 98.746} C_DIS
LIN {X -0.042,Y -477.117,Z 1186.546,A 0.000,B 0.000,C 90.000,E1 98.219} C_DIS
LIN {X 0.103,Y -475.621,Z 1186.543,A 0.000,B 0.000,C 90.000,E1 97.701} C_DIS
LIN {X -0.030,Y -474.407,Z 1186.542,A 0.000,B 0.000,C 90.000,E1 97.466} C_DIS
LIN {X -0.224,Y -472.791,Z 1186.540,A 0.000,B 0.000,C 90.000,E1 97.239} C_DIS
LIN {X 0.162,Y -458.271,Z 1186.529,A 0.000,B 0.000,C 90.000,E1 95.163} C_DIS
LIN {X 0.086,Y -440.597,Z 1186.514,A 0.000,B 0.000,C 90.000,E1 92.579} C_DIS
LIN {X 0.049,Y -422.820,Z 1186.498,A 0.000,B 0.000,C 90.000,E1 89.656} C_DIS
LIN {X 0.063,Y -411.065,Z 1186.486,A 0.000,B 0.000,C 90.000,E1 87.478} C_DIS
LIN {X 0.173,Y -400.744,Z 1186.475,A 0.000,B 0.000,C 90.000,E1 85.527} C_DIS
LIN {X 0.146,Y -389.062,Z 1186.463,A 0.000,B 0.000,C 90.000,E1 83.280} C_DIS
LIN {X -0.098,Y -380.329,Z 1186.453,A 0.000,B 0.000,C 90.000,E1 81.602} C_DIS
LIN {X -0.062,Y -371.311,Z 1186.444,A 0.000,B 0.000,C 90.000,E1 79.859} C_DIS
LIN {X -0.120,Y -361.986,Z 1186.434,A 0.000,B 0.000,C 90.000,E1 78.105} C_DIS
LIN {X -0.005,Y -352.429,Z 1186.424,A 0.000,B 0.000,C 90.000,E1 76.297} C_DIS
LIN {X 0.088,Y -341.136,Z 1186.412,A 0.000,B 0.000,C 90.000,E1 74.157} C_DIS
LIN {X 0.014,Y -328.397,Z 1186.398,A 0.000,B 0.000,C 90.000,E1 71.692} C_DIS
LIN {X -0.024,Y -314.577,Z 1186.382,A 0.000,B 0.000,C 90.000,E1 68.847} C_DIS
LIN {X -0.100,Y -300.143,Z 1186.364,A 0.000,B 0.000,C 90.000,E1 65.613} C_DIS
LIN {X -0.085,Y -288.055,Z 1186.348,A 0.000,B 0.000,C 90.000,E1 62.615} C_DIS
LIN {X -0.053,Y -275.419,Z 1186.329,A 0.000,B 0.000,C 90.000,E1 59.203} C_DIS
LIN {X -0.134,Y -264.662,Z 1186.311,A 0.000,B 0.000,C 90.000,E1 56.087} C_DIS
LIN {X 0.072,Y -254.446,Z 1186.294,A 0.000,B 0.000,C 90.000,E1 52.844} C_DIS
LIN {X -0.085,Y -244.853,Z 1186.276,A 0.000,B 0.000,C 90.000,E1 49.622} C_DIS
LIN {X 0.089,Y -234.798,Z 1186.255,A 0.000,B 0.000,C 90.000,E1 45.891} C_DIS
LIN {X -0.053,Y -225.627,Z 1186.234,A 0.000,B 0.000,C 90.000,E1 42.162} C_DIS
LIN {X 0.053,Y -218.893,Z 1186.217,A 0.000,B 0.000,C 90.000,E1 39.072} C_DIS
LIN {X 0.044,Y -211.287,Z 1186.196,A 0.000,B 0.000,C 90.000,E1 35.185} C_DIS
LIN {X -0.048,Y -204.552,Z 1186.174,A 0.000,B 0.000,C 90.000,E1 31.258} C_DIS
LIN {X -0.070,Y -198.469,Z 1186.151,A 0.000,B 0.000,C 90.000,E1 27.257} C_DIS
LIN {X -0.038,Y -194.126,Z 1186.133,A 0.000,B 0.000,C 90.000,E1 24.003} C_DIS
LIN {X 0.025,Y -189.501,Z 1186.110,A 0.000,B 0.000,C 90.000,E1 19.885} C_DIS
LIN {X 0.064,Y -185.755,Z 1186.088,A 0.000,B 0.000,C 90.000,E1 15.733} C_DIS
LIN {X 0.048,Y -182.583,Z 1186.060,A 0.000,B 0.000,C 90.000,E1 10.725} C_DIS
LIN {X 0.040,Y -180.514,Z 1186.018,A 0.000,B 0.000,C 90.000,E1 3.154} C_DIS
LIN {X -0.046,Y -182.203,Z 1185.969,A 0.000,B 0.000,C 90.000,E1 354.489} C_DIS
LIN {X -0.047,Y -185.208,Z 1185.941,A 0.000,B 0.000,C 90.000,E1 349.454} C_DIS
LIN {X -0.033,Y -188.779,Z 1185.918,A 0.000,B 0.000,C 90.000,E1 345.283} C_DIS
LIN {X -0.024,Y -193.320,Z 1185.895,A 0.000,B 0.000,C 90.000,E1 341.148} C_DIS
LIN {X 0.010,Y -198.537,Z 1185.873,A 0.000,B 0.000,C 90.000,E1 337.050} C_DIS
LIN {X 0.044,Y -204.344,Z 1185.850,A 0.000,B 0.000,C 90.000,E1 332.999} C_DIS
LIN {X 0.098,Y -210.814,Z 1185.828,A 0.000,B 0.000,C 90.000,E1 328.997} C_DIS
LIN {X -0.028,Y -216.487,Z 1185.810,A 0.000,B 0.000,C 90.000,E1 325.881} C_DIS
LIN {X 0.020,Y -224.020,Z 1185.789,A 0.000,B 0.000,C 90.000,E1 321.984} C_DIS
LIN {X -0.022,Y -231.014,Z 1185.772,A 0.000,B 0.000,C 90.000,E1 318.933} C_DIS
LIN {X 0.084,Y -239.078,Z 1185.755,A 0.000,B 0.000,C 90.000,E1 315.891} C_DIS
LIN {X 0.078,Y -248.312,Z 1185.739,A 0.000,B 0.000,C 90.000,E1 312.933} C_DIS
LIN {X -0.003,Y -259.971,Z 1185.720,A 0.000,B 0.000,C 90.000,E1 309.688} C_DIS
LIN {X -0.021,Y -272.825,Z 1185.703,A 0.000,B 0.000,C 90.000,E1 306.503} C_DIS
LIN {X 0.016,Y -284.136,Z 1185.689,A 0.000,B 0.000,C 90.000,E1 304.072} C_DIS
LIN {X 0.157,Y -296.688,Z 1185.676,A 0.000,B 0.000,C 90.000,E1 301.671} C_DIS
LIN {X -0.107,Y -312.626,Z 1185.661,A 0.000,B 0.000,C 90.000,E1 299.077} C_DIS
LIN {X -0.029,Y -325.996,Z 1185.651,A 0.000,B 0.000,C 90.000,E1 297.129} C_DIS
LIN {X 0.177,Y -335.783,Z 1185.644,A 0.000,B 0.000,C 90.000,E1 295.848} C_DIS
LIN {X 0.082,Y -354.007,Z 1185.632,A 0.000,B 0.000,C 90.000,E1 293.770} C_DIS
LIN {X -0.065,Y -380.724,Z 1185.617,A 0.000,B 0.000,C 90.000,E1 291.046} C_DIS
LIN {X -0.071,Y -394.328,Z 1185.610,A 0.000,B 0.000,C 90.000,E1 289.758} C_DIS
LIN {X -0.129,Y -407.628,Z 1185.603,A 0.000,B 0.000,C 90.000,E1 288.489} C_DIS
LIN {X 0.080,Y -415.278,Z 1185.598,A 0.000,B 0.000,C 90.000,E1 287.692} C_DIS
LIN {X 0.160,Y -425.311,Z 1185.592,A 0.000,B 0.000,C 90.000,E1 286.622} C_DIS
LIN {X 0.130,Y -434.801,Z 1185.587,A 0.000,B 0.000,C 90.000,E1 285.552} C_DIS
LIN {X -0.024,Y -441.273,Z 1185.582,A 0.000,B 0.000,C 90.000,E1 284.773} C_DIS
LIN {X -0.245,Y -447.023,Z 1185.578,A 0.000,B 0.000,C 90.000,E1 284.008} C_DIS
LIN {X 0.134,Y -452.103,Z 1185.573,A 0.000,B 0.000,C 90.000,E1 283.175} C_DIS
LIN {X 0.009,Y -456.524,Z 1185.569,A 0.000,B 0.000,C 90.000,E1 282.411} C_DIS
LIN {X -0.168,Y -460.221,Z 1185.565,A 0.000,B 0.000,C 90.000,E1 281.658} C_DIS
LIN {X -0.222,Y -463.297,Z 1185.560,A 0.000,B 0.000,C 90.000,E1 280.894} C_DIS
LIN {X -0.045,Y -466.462,Z 1185.555,A 0.000,B 0.000,C 90.000,E1 279.849} C_DIS
LIN {X 0.177,Y -468.989,Z 1185.549,A 0.000,B 0.000,C 90.000,E1 278.803} C_DIS
LIN {X -0.200,Y -469.940,Z 1185.546,A 0.000,B 0.000,C 90.000,E1 278.341} C_DIS
LIN {X -0.040,Y -470.610,Z 1185.543,A 0.000,B 0.000,C 90.000,E1 277.814} C_DIS
LIN {X 0.062,Y -470.927,Z 1185.541,A 0.000,B 0.000,C 90.000,E1 277.296} C_DIS
LIN {X 0.166,Y -470.857,Z 1185.538,A 0.000,B 0.000,C 90.000,E1 276.777} C_DIS
LIN {X -0.193,Y -470.330,Z 1185.535,A 0.000,B 0.000,C 90.000,E1 276.315} C_DIS
LIN {X -0.085,Y -469.350,Z 1185.532,A 0.000,B 0.000,C 90.000,E1 275.796} C_DIS
LIN {X 0.017,Y -467.918,Z 1185.529,A 0.000,B 0.000,C 90.000,E1 275.277} C_DIS
LIN {X 0.112,Y -466.100,Z 1185.526,A 0.000,B 0.000,C 90.000,E1 274.759} C_DIS
LIN {X 0.162,Y -463.725,Z 1185.524,A 0.000,B 0.000,C 90.000,E1 274.245} C_DIS
LIN {X 0.230,Y -460.711,Z 1185.521,A 0.000,B 0.000,C 90.000,E1 273.726} C_DIS
LIN {X -0.204,Y -456.806,Z 1185.518,A 0.000,B 0.000,C 90.000,E1 273.269} C_DIS
LIN {X 0.050,Y -454.499,Z 1185.517,A 0.000,B 0.000,C 90.000,E1 272.980} C_DIS
LIN {X 0.136,Y -449.067,Z 1185.514,A 0.000,B 0.000,C 90.000,E1 272.465} C_DIS
LIN {X -0.006,Y -445.906,Z 1185.512,A 0.000,B 0.000,C 90.000,E1 272.236} C_DIS
LIN {X 0.116,Y -442.761,Z 1185.511,A 0.000,B 0.000,C 90.000,E1 272.007} C_DIS
LIN {X -0.198,Y -435.943,Z 1185.509,A 0.000,B 0.000,C 90.000,E1 271.661} C_DIS
LIN {X 0.039,Y -428.899,Z 1185.507,A 0.000,B 0.000,C 90.000,E1 271.318} C_DIS
LIN {X -0.169,Y -421.985,Z 1185.506,A 0.000,B 0.000,C 90.000,E1 271.088} C_DIS
LIN {X -0.023,Y -411.584,Z 1185.504,A 0.000,B 0.000,C 90.000,E1 270.745} C_DIS
LIN {X 0.143,Y -400.989,Z 1185.503,A 0.000,B 0.000,C 90.000,E1 270.458} C_DIS
LIN {X -0.156,Y -389.949,Z 1185.501,A 0.000,B 0.000,C 90.000,E1 270.286} C_DIS
LIN {X -0.162,Y -381.782,Z 1185.501,A 0.000,B 0.000,C 90.000,E1 270.172} C_DIS
LIN {X 0.130,Y -373.570,Z 1185.500,A 0.000,B 0.000,C 90.000,E1 270.057} C_DIS
LIN {X -0.021,Y -367.935,Z 1185.500,A 0.000,B 0.000,C 90.000,E1 270.057} C_DIS
LIN {X -0.034,Y -181.567,Z 1185.500,A 0.000,B 0.000,C 90.000,E1 270.057} C_DIS
LIN {X -0.027,Y -180.848,Z 1185.472,A 0.000,B 0.000,C 90.000,E1 264.951} C_DIS
LIN {X 0.057,Y -178.958,Z 1185.444,A 0.000,B 0.000,C 90.000,E1 259.859} C_DIS
LIN {X -0.052,Y -177.360,Z 1185.430,A 0.000,B 0.000,C 90.000,E1 257.353} C_DIS
LIN {X 0.044,Y -175.533,Z 1185.411,A 0.000,B 0.000,C 90.000,E1 253.921} C_DIS
LIN {X 0.045,Y -172.267,Z 1185.387,A 0.000,B 0.000,C 90.000,E1 249.645} C_DIS
LIN {X 0.084,Y -171.747,Z 1185.382,A 0.000,B 0.000,C 90.000,E1 248.773} C_DIS
LIN {X -0.058,Y -167.344,Z 1185.353,A 0.000,B 0.000,C 90.000,E1 243.640} C_DIS
LIN {X 0.023,Y -166.731,Z 1185.349,A 0.000,B 0.000,C 90.000,E1 242.743} C_DIS
LIN {X -0.063,Y -162.711,Z 1185.324,A 0.000,B 0.000,C 90.000,E1 238.408} C_DIS
LIN {X -0.002,Y -161.402,Z 1185.315,A 0.000,B 0.000,C 90.000,E1 236.628} C_DIS
LIN {X 0.039,Y -157.395,Z 1185.290,A 0.000,B 0.000,C 90.000,E1 232.190} C_DIS
LIN {X -0.028,Y -155.392,Z 1185.275,A 0.000,B 0.000,C 90.000,E1 229.542} C_DIS
LIN {X 0.012,Y -151.726,Z 1185.250,A 0.000,B 0.000,C 90.000,E1 225.040} C_DIS
LIN {X 0.028,Y -149.920,Z 1185.235,A 0.000,B 0.000,C 90.000,E1 222.324} C_DIS
LIN {X -0.054,Y -146.773,Z 1185.210,A 0.000,B 0.000,C 90.000,E1 217.810} C_DIS
LIN {X 0.050,Y -145.344,Z 1185.195,A 0.000,B 0.000,C 90.000,E1 215.025} C_DIS
LIN {X -0.035,Y -142.419,Z 1185.164,A 0.000,B 0.000,C 90.000,E1 209.539} C_DIS
LIN {X 0.014,Y -141.406,Z 1185.149,A 0.000,B 0.000,C 90.000,E1 206.744} C_DIS
LIN {X 0.002,Y -139.357,Z 1185.113,A 0.000,B 0.000,C 90.000,E1 200.248} C_DIS
LIN {X -0.011,Y -138.798,Z 1185.097,A 0.000,B 0.000,C 90.000,E1 197.457} C_DIS
LIN {X 0.044,Y -138.348,Z 1185.055,A 0.000,B 0.000,C 90.000,E1 189.962} C_DIS
LIN {X 0.062,Y -139.371,Z 1185.009,A 0.000,B 0.000,C 90.000,E1 181.547} C_DIS
LIN {X -0.024,Y -141.260,Z 1184.973,A 0.000,B 0.000,C 90.000,E1 175.065} C_DIS
LIN {X -0.067,Y -142.627,Z 1184.957,A 0.000,B 0.000,C 90.000,E1 172.299} C_DIS
LIN {X 0.027,Y -144.950,Z 1184.931,A 0.000,B 0.000,C 90.000,E1 167.645} C_DIS
LIN {X 0.018,Y -147.579,Z 1184.911,A 0.000,B 0.000,C 90.000,E1 163.976} C_DIS
LIN {X 0.048,Y -150.191,Z 1184.891,A 0.000,B 0.000,C 90.000,E1 160.315} C_DIS
LIN {X -0.085,Y -153.571,Z 1184.871,A 0.000,B 0.000,C 90.000,E1 156.741} C_DIS
LIN {X -0.034,Y -156.988,Z 1184.851,A 0.000,B 0.000,C 90.000,E1 153.127} C_DIS
LIN {X 0.039,Y -161.102,Z 1184.831,A 0.000,B 0.000,C 90.000,E1 149.537} C_DIS
LIN {X -0.015,Y -163.205,Z 1184.821,A 0.000,B 0.000,C 90.000,E1 147.788} C_DIS
LIN {X -0.011,Y -167.633,Z 1184.802,A 0.000,B 0.000,C 90.000,E1 144.276} C_DIS
LIN {X 0.004,Y -171.458,Z 1184.787,A 0.000,B 0.000,C 90.000,E1 141.662} C_DIS
LIN {X -0.065,Y -176.384,Z 1184.768,A 0.000,B 0.000,C 90.000,E1 138.243} C_DIS
LIN {X 0.056,Y -180.677,Z 1184.754,A 0.000,B 0.000,C 90.000,E1 135.648} C_DIS
LIN {X 0.039,Y -186.079,Z 1184.735,A 0.000,B 0.000,C 90.000,E1 132.285} C_DIS
LIN {X -0.024,Y -190.716,Z 1184.721,A 0.000,B 0.000,C 90.000,E1 129.806} C_DIS
LIN {X 0.007,Y -196.469,Z 1184.703,A 0.000,B 0.000,C 90.000,E1 126.503} C_DIS
LIN {X -0.039,Y -201.310,Z 1184.689,A 0.000,B 0.000,C 90.000,E1 124.040} C_DIS
LIN {X 0.144,Y -311.537,Z 1184.689,A 0.000,B 0.000,C 90.000,E1 123.992} C_DIS
LIN {X 0.039,Y -312.661,Z 1184.689,A 0.000,B 0.000,C 90.000,E1 123.992} C_DIS
LIN {X 0.154,Y -317.002,Z 1184.688,A 0.000,B 0.000,C 90.000,E1 123.785} C_DIS
LIN {X 0.006,Y -319.403,Z 1184.687,A 0.000,B 0.000,C 90.000,E1 123.627} C_DIS
LIN {X 0.062,Y -322.666,Z 1184.685,A 0.000,B 0.000,C 90.000,E1 123.245} C_DIS
LIN {X -0.057,Y -324.596,Z 1184.683,A 0.000,B 0.000,C 90.000,E1 122.959} C_DIS
LIN {X 0.096,Y -326.102,Z 1184.681,A 0.000,B 0.000,C 90.000,E1 122.625} C_DIS
LIN {X -0.084,Y -339.473,Z 1184.662,A 0.000,B 0.000,C 90.000,E1 119.205} C_DIS
LIN {X 0.091,Y -351.863,Z 1184.647,A 0.000,B 0.000,C 90.000,E1 116.411} C_DIS
LIN {X 0.163,Y -365.748,Z 1184.632,A 0.000,B 0.000,C 90.000,E1 113.695} C_DIS
LIN {X 0.083,Y -379.445,Z 1184.619,A 0.000,B 0.000,C 90.000,E1 111.354} C_DIS
LIN {X -0.151,Y -394.518,Z 1184.606,A 0.000,B 0.000,C 90.000,E1 109.087} C_DIS
LIN {X 0.105,Y -411.073,Z 1184.593,A 0.000,B 0.000,C 90.000,E1 106.804} C_DIS
LIN {X -0.146,Y -429.225,Z 1184.581,A 0.000,B 0.000,C 90.000,E1 104.647} C_DIS
LIN {X -0.116,Y -448.875,Z 1184.570,A 0.000,B 0.000,C 90.000,E1 102.535} C_DIS
LIN {X -0.213,Y -469.204,Z 1184.559,A 0.000,B 0.000,C 90.000,E1 100.602} C_DIS
LIN {X -0.189,Y -471.561,Z 1184.557,A 0.000,B 0.000,C 90.000,E1 100.366} C_DIS
LIN {X 0.195,Y -473.425,Z 1184.556,A 0.000,B 0.000,C 90.000,E1 100.074} C_DIS
LIN {X 0.032,Y -474.834,Z 1184.555,A 0.000,B 0.000,C 90.000,E1 99.849} C_DIS
LIN {X 0.229,Y -476.694,Z 1184.552,A 0.000,B 0.000,C 90.000,E1 99.321} C_DIS
LIN {X -0.116,Y -477.452,Z 1184.549,A 0.000,B 0.000,C 90.000,E1 98.859} C_DIS
LIN {X 0.025,Y -477.234,Z 1184.546,A 0.000,B 0.000,C 90.000,E1 98.341} C_DIS
LIN {X 0.236,Y -476.012,Z 1184.544,A 0.000,B 0.000,C 90.000,E1 97.814} C_DIS
LIN {X 0.041,Y -474.969,Z 1184.542,A 0.000,B 0.000,C 90.000,E1 97.587} C_DIS
LIN {X -0.092,Y -473.566,Z 1184.541,A 0.000,B 0.000,C 90.000,E1 97.352} C_DIS
LIN {X -0.153,Y -459.088,Z 1184.530,A 0.000,B 0.000,C 90.000,E1 95.334} C_DIS
LIN {X -0.197,Y -441.381,Z 1184.515,A 0.000,B 0.000,C 90.000,E1 92.751} C_DIS
LIN {X -0.201,Y -423.509,Z 1184.499,A 0.000,B 0.000,C 90.000,E1 89.828} C_DIS
LIN {X -0.077,Y -410.250,Z 1184.485,A 0.000,B 0.000,C 90.000,E1 87.364} C_DIS
LIN {X 0.014,Y -399.922,Z 1184.474,A 0.000,B 0.000,C 90.000,E1 85.412} C_DIS
LIN {X -0.031,Y -388.223,Z 1184.462,A 0.000,B 0.000,C 90.000,E1 83.166} C_DIS
LIN {X 0.087,Y -379.469,Z 1184.453,A 0.000,B 0.000,C 90.000,E1 81.432} C_DIS
LIN {X 0.098,Y -370.431,Z 1184.443,A 0.000,B 0.000,C 90.000,E1 79.690} C_DIS
LIN {X 0.014,Y -361.075,Z 1184.433,A 0.000,B 0.000,C 90.000,E1 77.937} C_DIS
LIN {X -0.156,Y -351.515,Z 1184.423,A 0.000,B 0.000,C 90.000,E1 76.172} C_DIS
LIN {X -0.068,Y -340.225,Z 1184.411,A 0.000,B 0.000,C 90.000,E1 74.031} C_DIS
LIN {X 0.055,Y -327.484,Z 1184.397,A 0.000,B 0.000,C 90.000,E1 71.529} C_DIS
LIN {X 0.014,Y -312.232,Z 1184.380,A 0.000,B 0.000,C 90.000,E1 68.358} C_DIS
LIN {X -0.133,Y -296.587,Z 1184.360,A 0.000,B 0.000,C 90.000,E1 64.793} C_DIS
LIN {X -0.081,Y -284.690,Z 1184.343,A 0.000,B 0.000,C 90.000,E1 61.769} C_DIS
LIN {X 0.043,Y -273.432,Z 1184.326,A 0.000,B 0.000,C 90.000,E1 58.663} C_DIS
LIN {X 0.052,Y -262.749,Z 1184.308,A 0.000,B 0.000,C 90.000,E1 55.515} C_DIS
LIN {X -0.126,Y -251.511,Z 1184.289,A 0.000,B 0.000,C 90.000,E1 51.984} C_DIS
LIN {X -0.042,Y -243.096,Z 1184.272,A 0.000,B 0.000,C 90.000,E1 49.057} C_DIS
LIN {X 0.082,Y -233.146,Z 1184.252,A 0.000,B 0.000,C 90.000,E1 45.324} C_DIS
LIN {X 0.057,Y -224.118,Z 1184.231,A 0.000,B 0.000,C 90.000,E1 41.553} C_DIS
LIN {X -0.035,Y -215.939,Z 1184.210,A 0.000,B 0.000,C 90.000,E1 37.729} C_DIS
LIN {X 0.078,Y -208.632,Z 1184.188,A 0.000,B 0.000,C 90.000,E1 33.785} C_DIS
LIN {X 0.036,Y -202.100,Z 1184.166,A 0.000,B 0.000,C 90.000,E1 29.823} C_DIS
LIN {X 0.025,Y -196.212,Z 1184.143,A 0.000,B 0.000,C 90.000,E1 25.796} C_DIS
LIN {X 0.022,Y -191.202,Z 1184.121,A 0.000,B 0.000,C 90.000,E1 21.716} C_DIS
LIN {X 0.046,Y -186.975,Z 1184.098,A 0.000,B 0.000,C 90.000,E1 17.583} C_DIS
LIN {X 0.021,Y -183.295,Z 1184.070,A 0.000,B 0.000,C 90.000,E1 12.591} C_DIS
LIN {X -0.006,Y -180.728,Z 1184.037,A 0.000,B 0.000,C 90.000,E1 6.720} C_DIS
LIN {X -0.058,Y -181.869,Z 1183.969,A 0.000,B 0.000,C 90.000,E1 354.489} C_DIS
LIN {X -0.071,Y -184.864,Z 1183.941,A 0.000,B 0.000,C 90.000,E1 349.454} C_DIS
LIN {X -0.069,Y -188.428,Z 1183.918,A 0.000,B 0.000,C 90.000,E1 345.283} C_DIS
LIN {X -0.073,Y -192.961,Z 1183.895,A 0.000,B 0.000,C 90.000,E1 341.148} C_DIS
LIN {X -0.052,Y -198.175,Z 1183.872,A 0.000,B 0.000,C 90.000,E1 337.050} C_DIS
LIN {X -0.029,Y -203.993,Z 1183.850,A 0.000,B 0.000,C 90.000,E1 332.999} C_DIS
LIN {X 0.010,Y -210.500,Z 1183.828,A 0.000,B 0.000,C 90.000,E1 328.997} C_DIS
LIN {X 0.040,Y -217.633,Z 1183.806,A 0.000,B 0.000,C 90.000,E1 325.055} C_DIS
LIN {X -0.091,Y -223.744,Z 1183.789,A 0.000,B 0.000,C 90.000,E1 321.984} C_DIS
LIN {X -0.143,Y -230.785,Z 1183.772,A 0.000,B 0.000,C 90.000,E1 318.933} C_DIS
LIN {X -0.041,Y -238.914,Z 1183.755,A 0.000,B 0.000,C 90.000,E1 315.891} C_DIS
LIN {X -0.055,Y -248.200,Z 1183.738,A 0.000,B 0.000,C 90.000,E1 312.933} C_DIS
LIN {X 0.054,Y -259.890,Z 1183.720,A 0.000,B 0.000,C 90.000,E1 309.644} C_DIS
LIN {X 0.046,Y -272.822,Z 1183.703,A 0.000,B 0.000,C 90.000,E1 306.457} C_DIS
LIN {X 0.016,Y -284.149,Z 1183.689,A 0.000,B 0.000,C 90.000,E1 304.040} C_DIS
LIN {X -0.008,Y -296.780,Z 1183.676,A 0.000,B 0.000,C 90.000,E1 301.671} C_DIS
LIN {X -0.004,Y -312.749,Z 1183.661,A 0.000,B 0.000,C 90.000,E1 299.027} C_DIS
LIN {X 0.156,Y -323.776,Z 1183.652,A 0.000,B 0.000,C 90.000,E1 297.385} C_DIS
LIN {X -0.028,Y -333.406,Z 1183.645,A 0.000,B 0.000,C 90.000,E1 296.155} C_DIS
LIN {X 0.103,Y -353.787,Z 1183.632,A 0.000,B 0.000,C 90.000,E1 293.770} C_DIS
LIN {X -0.137,Y -380.669,Z 1183.617,A 0.000,B 0.000,C 90.000,E1 291.046} C_DIS
LIN {X -0.092,Y -396.935,Z 1183.608,A 0.000,B 0.000,C 90.000,E1 289.504} C_DIS
LIN {X -0.101,Y -410.111,Z 1183.601,A 0.000,B 0.000,C 90.000,E1 288.236} C_DIS
LIN {X -0.087,Y -417.721,Z 1183.597,A 0.000,B 0.000,C 90.000,E1 287.457} C_DIS
LIN {X 0.027,Y -427.568,Z 1183.591,A 0.000,B 0.000,C 90.000,E1 286.386} C_DIS
LIN {X -0.121,Y -434.605,Z 1183.587,A 0.000,B 0.000,C 90.000,E1 285.607} C_DIS
LIN {X 0.144,Y -441.079,Z 1183.582,A 0.000,B 0.000,C 90.000,E1 284.773} C_DIS
LIN {X -0.076,Y -446.878,Z 1183.578,A 0.000,B 0.000,C 90.000,E1 284.008} C_DIS
LIN {X -0.136,Y -451.958,Z 1183.573,A 0.000,B 0.000,C 90.000,E1 283.231} C_DIS
LIN {X 0.179,Y -456.423,Z 1183.569,A 0.000,B 0.000,C 90.000,E1 282.411} C_DIS
LIN {X 0.002,Y -460.197,Z 1183.565,A 0.000,B 0.000,C 90.000,E1 281.658} C_DIS
LIN {X -0.051,Y -463.299,Z 1183.561,A 0.000,B 0.000,C 90.000,E1 280.894} C_DIS
LIN {X 0.128,Y -466.596,Z 1183.555,A 0.000,B 0.000,C 90.000,E1 279.849} C_DIS
LIN {X -0.113,Y -469.211,Z 1183.549,A 0.000,B 0.000,C 90.000,E1 278.859} C_DIS
LIN {X -0.024,Y -470.198,Z 1183.546,A 0.000,B 0.000,C 90.000,E1 278.341} C_DIS
LIN {X 0.139,Y -470.883,Z 1183.543,A 0.000,B 0.000,C 90.000,E1 277.814} C_DIS
LIN {X 0.241,Y -471.204,Z 1183.541,A 0.000,B 0.000,C 90.000,E1 277.296} C_DIS
LIN {X -0.121,Y -471.156,Z 1183.538,A 0.000,B 0.000,C 90.000,E1 276.834} C_DIS
LIN {X -0.011,Y -470.659,Z 1183.535,A 0.000,B 0.000,C 90.000,E1 276.315} C_DIS
LIN {X 0.098,Y -469.671,Z 1183.532,A 0.000,B 0.000,C 90.000,E1 275.796} C_DIS
LIN {X 0.202,Y -468.246,Z 1183.529,A 0.000,B 0.000,C 90.000,E1 275.277} C_DIS
LIN {X -0.205,Y -466.446,Z 1183.527,A 0.000,B 0.000,C 90.000,E1 274.821} C_DIS
LIN {X -0.114,Y -464.139,Z 1183.524,A 0.000,B 0.000,C 90.000,E1 274.302} C_DIS
LIN {X -0.042,Y -461.177,Z 1183.521,A 0.000,B 0.000,C 90.000,E1 273.784} C_DIS
LIN {X -0.015,Y -457.345,Z 1183.518,A 0.000,B 0.000,C 90.000,E1 273.269} C_DIS
LIN {X 0.017,Y -452.478,Z 1183.515,A 0.000,B 0.000,C 90.000,E1 272.751} C_DIS
LIN {X -0.155,Y -449.720,Z 1183.514,A 0.000,B 0.000,C 90.000,E1 272.522} C_DIS
LIN {X -0.189,Y -443.455,Z 1183.511,A 0.000,B 0.000,C 90.000,E1 272.064} C_DIS
LIN {X -0.064,Y -436.799,Z 1183.509,A 0.000,B 0.000,C 90.000,E1 271.661} C_DIS
LIN {X 0.121,Y -429.740,Z 1183.507,A 0.000,B 0.000,C 90.000,E1 271.318} C_DIS
LIN {X -0.146,Y -422.750,Z 1183.506,A 0.000,B 0.000,C 90.000,E1 271.088} C_DIS
LIN {X -0.055,Y -412.207,Z 1183.504,A 0.000,B 0.000,C 90.000,E1 270.745} C_DIS
LIN {X 0.102,Y -401.551,Z 1183.503,A 0.000,B 0.000,C 90.000,E1 270.458} C_DIS
LIN {X -0.191,Y -390.550,Z 1183.501,A 0.000,B 0.000,C 90.000,E1 270.286} C_DIS
LIN {X 0.186,Y -382.667,Z 1183.501,A 0.000,B 0.000,C 90.000,E1 270.115} C_DIS
LIN {X 0.085,Y -374.924,Z 1183.500,A 0.000,B 0.000,C 90.000,E1 270.057} C_DIS
LIN {X -0.119,Y -367.804,Z 1183.500,A 0.000,B 0.000,C 90.000,E1 270.057} C_DIS
LIN {X -0.083,Y -181.565,Z 1183.500,A 0.000,B 0.000,C 90.000,E1 270.057} C_DIS
LIN {X -0.057,Y -180.845,Z 1183.472,A 0.000,B 0.000,C 90.000,E1 264.951} C_DIS
LIN {X 0.025,Y -178.954,Z 1183.444,A 0.000,B 0.000,C 90.000,E1 259.859} C_DIS
LIN {X -0.083,Y -177.355,Z 1183.430,A 0.000,B 0.000,C 90.000,E1 257.353} C_DIS
LIN {X 0.014,Y -175.525,Z 1183.411,A 0.000,B 0.000,C 90.000,E1 253.921} C_DIS
LIN {X 0.016,Y -172.261,Z 1183.387,A 0.000,B 0.000,C 90.000,E1 249.645} C_DIS
LIN {X 0.054,Y -171.740,Z 1183.382,A 0.000,B 0.000,C 90.000,E1 248.773} C_DIS
LIN {X -0.088,Y -167.337,Z 1183.353,A 0.000,B 0.000,C 90.000,E1 243.640} C_DIS
LIN {X -0.006,Y -166.723,Z 1183.349,A 0.000,B 0.000,C 90.000,E1 242.743} C_DIS
LIN {X -0.008,Y -162.703,Z 1183.324,A 0.000,B 0.000,C 90.000,E1 238.377} C_DIS
LIN {X -0.031,Y -161.394,Z 1183.315,A 0.000,B 0.000,C 90.000,E1 236.628} C_DIS
LIN {X 0.011,Y -157.386,Z 1183.290,A 0.000,B 0.000,C 90.000,E1 232.190} C_DIS
LIN {X -0.055,Y -155.382,Z 1183.275,A 0.000,B 0.000,C 90.000,E1 229.542} C_DIS
LIN {X -0.015,Y -151.718,Z 1183.250,A 0.000,B 0.000,C 90.000,E1 225.040} C_DIS
LIN {X 0.000,Y -149.911,Z 1183.235,A 0.000,B 0.000,C 90.000,E1 222.324} C_DIS
LIN {X -0.081,Y -146.767,Z 1183.210,A 0.000,B 0.000,C 90.000,E1 217.810} C_DIS
LIN {X 0.022,Y -145.336,Z 1183.195,A 0.000,B 0.000,C 90.000,E1 215.025} C_DIS
LIN {X -0.062,Y -142.415,Z 1183.164,A 0.000,B 0.000,C 90.000,E1 209.539} C_DIS
LIN {X -0.012,Y -141.400,Z 1183.149,A 0.000,B 0.000,C 90.000,E1 206.744} C_DIS
LIN {X -0.025,Y -139.356,Z 1183.112,A 0.000,B 0.000,C 90.000,E1 200.248} C_DIS
LIN {X -0.037,Y -138.795,Z 1183.097,A 0.000,B 0.000,C 90.000,E1 197.457} C_DIS
LIN {X 0.018,Y -138.347,Z 1183.055,A 0.000,B 0.000,C 90.000,E1 189.962} C_DIS
LIN {X 0.035,Y -139.375,Z 1183.009,A 0.000,B 0.000,C 90.000,E1 181.547} C_DIS
LIN {X -0.051,Y -141.265,Z 1182.972,A 0.000,B 0.000,C 90.000,E1 175.065} C_DIS
LIN {X 0.048,Y -142.631,Z 1182.957,A 0.000,B 0.000,C 90.000,E1 172.243} C_DIS
LIN {X 0.000,Y -144.957,Z 1182.931,A 0.000,B 0.000,C 90.000,E1 167.645} C_DIS
LIN {X -0.009,Y -147.586,Z 1182.911,A 0.000,B 0.000,C 90.000,E1 163.976} C_DIS
LIN {X 0.021,Y -150.200,Z 1182.891,A 0.000,B 0.000,C 90.000,E1 160.315} C_DIS
LIN {X 0.088,Y -153.583,Z 1182.871,A 0.000,B 0.000,C 90.000,E1 156.666} C_DIS
LIN {X -0.063,Y -156.999,Z 1182.851,A 0.000,B 0.000,C 90.000,E1 153.127} C_DIS
LIN {X 0.010,Y -161.115,Z 1182.831,A 0.000,B 0.000,C 90.000,E1 149.537} C_DIS
LIN {X -0.045,Y -163.217,Z 1182.821,A 0.000,B 0.000,C 90.000,E1 147.788} C_DIS
LIN {X -0.041,Y -167.647,Z 1182.802,A 0.000,B 0.000,C 90.000,E1 144.276} C_DIS
LIN {X -0.026,Y -171.472,Z 1182.787,A 0.000,B 0.000,C 90.000,E1 141.662} C_DIS
LIN {X -0.096,Y -176.399,Z 1182.768,A 0.000,B 0.000,C 90.000,E1 138.243} C_DIS
LIN {X 0.025,Y -180.694,Z 1182.754,A 0.000,B 0.000,C 90.000,E1 135.648} C_DIS
LIN {X 0.007,Y -186.096,Z 1182.735,A 0.000,B 0.000,C 90.000,E1 132.285} C_DIS
LIN {X -0.057,Y -190.734,Z 1182.721,A 0.000,B 0.000,C 90.000,E1 129.806} C_DIS
LIN {X -0.025,Y -196.487,Z 1182.703,A 0.000,B 0.000,C 90.000,E1 126.503} C_DIS
LIN {X 0.030,Y -201.276,Z 1182.689,A 0.000,B 0.000,C 90.000,E1 124.040} C_DIS
LIN {X 0.011,Y -311.270,Z 1182.689,A 0.000,B 0.000,C 90.000,E1 124.040} C_DIS
LIN {X -0.012,Y -313.689,Z 1182.689,A 0.000,B 0.000,C 90.000,E1 123.992} C_DIS
LIN {X 0.102,Y -317.378,Z 1182.688,A 0.000,B 0.000,C 90.000,E1 123.785} C_DIS
LIN {X -0.047,Y -319.646,Z 1182.687,A 0.000,B 0.000,C 90.000,E1 123.627} C_DIS
LIN {X 0.009,Y -322.795,Z 1182.685,A 0.000,B 0.000,C 90.000,E1 123.245} C_DIS
LIN {X -0.154,Y -324.715,Z 1182.683,A 0.000,B 0.000,C 90.000,E1 122.959} C_DIS
LIN {X -0.046,Y -326.205,Z 1182.681,A 0.000,B 0.000,C 90.000,E1 122.625} C_DIS
LIN {X 0.068,Y -339.552,Z 1182.662,A 0.000,B 0.000,C 90.000,E1 119.155} C_DIS
LIN {X -0.056,Y -351.956,Z 1182.647,A 0.000,B 0.000,C 90.000,E1 116.411} C_DIS
LIN {X 0.011,Y -365.854,Z 1182.632,A 0.000,B 0.000,C 90.000,E1 113.695} C_DIS
LIN {X -0.070,Y -379.564,Z 1182.619,A 0.000,B 0.000,C 90.000,E1 111.354} C_DIS
LIN {X 0.066,Y -394.651,Z 1182.606,A 0.000,B 0.000,C 90.000,E1 109.033} C_DIS
LIN {X -0.055,Y -411.221,Z 1182.593,A 0.000,B 0.000,C 90.000,E1 106.804} C_DIS
LIN {X 0.107,Y -429.390,Z 1182.581,A 0.000,B 0.000,C 90.000,E1 104.592} C_DIS
LIN {X 0.162,Y -449.051,Z 1182.569,A 0.000,B 0.000,C 90.000,E1 102.479} C_DIS
LIN {X 0.093,Y -469.384,Z 1182.559,A 0.000,B 0.000,C 90.000,E1 100.546} C_DIS
LIN {X 0.119,Y -471.679,Z 1182.557,A 0.000,B 0.000,C 90.000,E1 100.310} C_DIS
LIN {X 0.007,Y -473.514,Z 1182.556,A 0.000,B 0.000,C 90.000,E1 100.074} C_DIS
LIN {X -0.187,Y -474.898,Z 1182.555,A 0.000,B 0.000,C 90.000,E1 99.849} C_DIS
LIN {X 0.009,Y -476.680,Z 1182.552,A 0.000,B 0.000,C 90.000,E1 99.321} C_DIS
LIN {X 0.136,Y -477.374,Z 1182.549,A 0.000,B 0.000,C 90.000,E1 98.803} C_DIS
LIN {X -0.194,Y -477.095,Z 1182.546,A 0.000,B 0.000,C 90.000,E1 98.341} C_DIS
LIN {X 0.017,Y -475.807,Z 1182.543,A 0.000,B 0.000,C 90.000,E1 97.814} C_DIS
LIN {X -0.178,Y -474.720,Z 1182.542,A 0.000,B 0.000,C 90.000,E1 97.587} C_DIS
LIN {X 0.159,Y -473.268,Z 1182.541,A 0.000,B 0.000,C 90.000,E1 97.296} C_DIS
LIN {X 0.085,Y -458.787,Z 1182.529,A 0.000,B 0.000,C 90.000,E1 95.277} C_DIS
LIN {X 0.025,Y -441.118,Z 1182.515,A 0.000,B 0.000,C 90.000,E1 92.694} C_DIS
LIN {X 0.004,Y -423.260,Z 1182.499,A 0.000,B 0.000,C 90.000,E1 89.771} C_DIS
LIN {X 0.114,Y -409.984,Z 1182.485,A 0.000,B 0.000,C 90.000,E1 87.306} C_DIS
LIN {X -0.204,Y -399.670,Z 1182.474,A 0.000,B 0.000,C 90.000,E1 85.412} C_DIS
LIN {X 0.137,Y -387.938,Z 1182.462,A 0.000,B 0.000,C 90.000,E1 83.109} C_DIS
LIN {X -0.131,Y -379.169,Z 1182.452,A 0.000,B 0.000,C 90.000,E1 81.432} C_DIS
LIN {X -0.120,Y -370.137,Z 1182.443,A 0.000,B 0.000,C 90.000,E1 79.690} C_DIS
LIN {X 0.148,Y -360.763,Z 1182.433,A 0.000,B 0.000,C 90.000,E1 77.881} C_DIS
LIN {X -0.033,Y -351.197,Z 1182.423,A 0.000,B 0.000,C 90.000,E1 76.117} C_DIS
LIN {X 0.041,Y -339.919,Z 1182.411,A 0.000,B 0.000,C 90.000,E1 73.976} C_DIS
LIN {X -0.058,Y -327.157,Z 1182.397,A 0.000,B 0.000,C 90.000,E1 71.511} C_DIS
LIN {X -0.087,Y -311.942,Z 1182.380,A 0.000,B 0.000,C 90.000,E1 68.337} C_DIS
LIN {X 0.042,Y -297.665,Z 1182.361,A 0.000,B 0.000,C 90.000,E1 65.049} C_DIS
LIN {X 0.111,Y -285.690,Z 1182.345,A 0.000,B 0.000,C 90.000,E1 62.025} C_DIS
LIN {X -0.115,Y -274.358,Z 1182.328,A 0.000,B 0.000,C 90.000,E1 58.997} C_DIS
LIN {X 0.143,Y -263.600,Z 1182.310,A 0.000,B 0.000,C 90.000,E1 55.801} C_DIS
LIN {X -0.016,Y -252.277,Z 1182.290,A 0.000,B 0.000,C 90.000,E1 52.271} C_DIS
LIN {X -0.073,Y -242.757,Z 1182.272,A 0.000,B 0.000,C 90.000,E1 49.013} C_DIS
LIN {X 0.031,Y -232.804,Z 1182.252,A 0.000,B 0.000,C 90.000,E1 45.283} C_DIS
LIN {X -0.012,Y -223.824,Z 1182.231,A 0.000,B 0.000,C 90.000,E1 41.515} C_DIS
LIN {X 0.048,Y -215.660,Z 1182.209,A 0.000,B 0.000,C 90.000,E1 37.649} C_DIS
LIN {X -0.026,Y -208.336,Z 1182.188,A 0.000,B 0.000,C 90.000,E1 33.754} C_DIS
LIN {X -0.087,Y -201.754,Z 1182.165,A 0.000,B 0.000,C 90.000,E1 29.795} C_DIS
LIN {X 0.062,Y -195.860,Z 1182.143,A 0.000,B 0.000,C 90.000,E1 25.720} C_DIS
LIN {X -0.032,Y -190.821,Z 1182.120,A 0.000,B 0.000,C 90.000,E1 21.663} C_DIS
LIN {X 0.043,Y -186.610,Z 1182.097,A 0.000,B 0.000,C 90.000,E1 17.511} C_DIS
LIN {X -0.045,Y -182.938,Z 1182.070,A 0.000,B 0.000,C 90.000,E1 12.535} C_DIS
LIN {X -0.083,Y -180.369,Z 1182.037,A 0.000,B 0.000,C 90.000,E1 6.663} C_DIS
LIN {X -0.070,Y -181.537,Z 1181.969,A 0.000,B 0.000,C 90.000,E1 354.489} C_DIS
LIN {X 0.085,Y -184.515,Z 1181.941,A 0.000,B 0.000,C 90.000,E1 349.398} C_DIS
LIN {X 0.075,Y -188.081,Z 1181.918,A 0.000,B 0.000,C 90.000,E1 345.227} C_DIS
LIN {X 0.062,Y -192.587,Z 1181.895,A 0.000,B 0.000,C 90.000,E1 341.094} C_DIS
LIN {X -0.113,Y -197.813,Z 1181.872,A 0.000,B 0.000,C 90.000,E1 337.050} C_DIS
LIN {X -0.104,Y -203.646,Z 1181.850,A 0.000,B 0.000,C 90.000,E1 332.999} C_DIS
LIN {X -0.077,Y -210.183,Z 1181.828,A 0.000,B 0.000,C 90.000,E1 328.997} C_DIS
LIN {X -0.061,Y -217.310,Z 1181.806,A 0.000,B 0.000,C 90.000,E1 325.055} C_DIS
LIN {X 0.111,Y -223.463,Z 1181.789,A 0.000,B 0.000,C 90.000,E1 321.904} C_DIS
LIN {X 0.060,Y -230.550,Z 1181.771,A 0.000,B 0.000,C 90.000,E1 318.852} C_DIS
LIN {X -0.002,Y -238.750,Z 1181.755,A 0.000,B 0.000,C 90.000,E1 315.850} C_DIS
LIN {X -0.027,Y -248.082,Z 1181.738,A 0.000,B 0.000,C 90.000,E1 312.894} C_DIS
LIN {X -0.097,Y -259.821,Z 1181.720,A 0.000,B 0.000,C 90.000,E1 309.644} C_DIS
LIN {X 0.049,Y -272.823,Z 1181.702,A 0.000,B 0.000,C 90.000,E1 306.423} C_DIS
LIN {X 0.086,Y -284.169,Z 1181.689,A 0.000,B 0.000,C 90.000,E1 303.992} C_DIS
LIN {X -0.182,Y -296.881,Z 1181.676,A 0.000,B 0.000,C 90.000,E1 301.671} C_DIS
LIN {X -0.032,Y -312.883,Z 1181.661,A 0.000,B 0.000,C 90.000,E1 298.999} C_DIS
LIN {X -0.029,Y -323.894,Z 1181.652,A 0.000,B 0.000,C 90.000,E1 297.385} C_DIS
LIN {X 0.028,Y -336.102,Z 1181.643,A 0.000,B 0.000,C 90.000,E1 295.796} C_DIS
LIN {X 0.129,Y -354.229,Z 1181.632,A 0.000,B 0.000,C 90.000,E1 293.695} C_DIS
LIN {X -0.066,Y -378.491,Z 1181.618,A 0.000,B 0.000,C 90.000,E1 291.227} C_DIS
LIN {X -0.026,Y -394.595,Z 1181.609,A 0.000,B 0.000,C 90.000,E1 289.704} C_DIS
LIN {X -0.120,Y -407.699,Z 1181.603,A 0.000,B 0.000,C 90.000,E1 288.471} C_DIS
LIN {X 0.184,Y -417.843,Z 1181.597,A 0.000,B 0.000,C 90.000,E1 287.402} C_DIS
LIN {X 0.154,Y -425.216,Z 1181.592,A 0.000,B 0.000,C 90.000,E1 286.622} C_DIS
LIN {X 0.091,Y -434.809,Z 1181.586,A 0.000,B 0.000,C 90.000,E1 285.552} C_DIS
LIN {X -0.064,Y -441.287,Z 1181.582,A 0.000,B 0.000,C 90.000,E1 284.773} C_DIS
LIN {X 0.149,Y -447.068,Z 1181.578,A 0.000,B 0.000,C 90.000,E1 283.953} C_DIS
LIN {X 0.094,Y -452.130,Z 1181.573,A 0.000,B 0.000,C 90.000,E1 283.175} C_DIS
LIN {X -0.031,Y -456.587,Z 1181.569,A 0.000,B 0.000,C 90.000,E1 282.411} C_DIS
LIN {X -0.208,Y -460.371,Z 1181.565,A 0.000,B 0.000,C 90.000,E1 281.658} C_DIS
LIN {X 0.194,Y -463.483,Z 1181.560,A 0.000,B 0.000,C 90.000,E1 280.838} C_DIS
LIN {X -0.082,Y -466.857,Z 1181.555,A 0.000,B 0.000,C 90.000,E1 279.849} C_DIS
LIN {X 0.143,Y -469.512,Z 1181.549,A 0.000,B 0.000,C 90.000,E1 278.803} C_DIS
LIN {X -0.231,Y -470.509,Z 1181.546,A 0.000,B 0.000,C 90.000,E1 278.341} C_DIS
LIN {X -0.067,Y -471.176,Z 1181.543,A 0.000,B 0.000,C 90.000,E1 277.814} C_DIS
LIN {X 0.036,Y -471.486,Z 1181.541,A 0.000,B 0.000,C 90.000,E1 277.296} C_DIS
LIN {X 0.146,Y -471.411,Z 1181.538,A 0.000,B 0.000,C 90.000,E1 276.777} C_DIS
LIN {X -0.212,Y -470.871,Z 1181.535,A 0.000,B 0.000,C 90.000,E1 276.315} C_DIS
LIN {X -0.101,Y -469.886,Z 1181.532,A 0.000,B 0.000,C 90.000,E1 275.796} C_DIS
LIN {X 0.005,Y -468.457,Z 1181.529,A 0.000,B 0.000,C 90.000,E1 275.277} C_DIS
LIN {X -0.102,Y -465.546,Z 1181.525,A 0.000,B 0.000,C 90.000,E1 274.531} C_DIS
LIN {X -0.022,Y -462.878,Z 1181.522,A 0.000,B 0.000,C 90.000,E1 274.012} C_DIS
LIN {X 0.228,Y -461.322,Z 1181.521,A 0.000,B 0.000,C 90.000,E1 273.726} C_DIS
LIN {X -0.203,Y -457.514,Z 1181.518,A 0.000,B 0.000,C 90.000,E1 273.269} C_DIS
LIN {X -0.168,Y -452.613,Z 1181.515,A 0.000,B 0.000,C 90.000,E1 272.751} C_DIS
LIN {X 0.115,Y -449.800,Z 1181.514,A 0.000,B 0.000,C 90.000,E1 272.465} C_DIS
LIN {X 0.082,Y -443.513,Z 1181.511,A 0.000,B 0.000,C 90.000,E1 272.007} C_DIS
LIN {X 0.190,Y -436.806,Z 1181.509,A 0.000,B 0.000,C 90.000,E1 271.604} C_DIS
LIN {X -0.066,Y -429.753,Z 1181.507,A 0.000,B 0.000,C 90.000,E1 271.318} C_DIS
LIN {X 0.098,Y -422.771,Z 1181.506,A 0.000,B 0.000,C 90.000,E1 271.031} C_DIS
LIN {X 0.189,Y -412.082,Z 1181.504,A 0.000,B 0.000,C 90.000,E1 270.688} C_DIS
LIN {X 0.014,Y -401.814,Z 1181.503,A 0.000,B 0.000,C 90.000,E1 270.458} C_DIS
LIN {X 0.157,Y -391.122,Z 1181.501,A 0.000,B 0.000,C 90.000,E1 270.229} C_DIS
LIN {X 0.135,Y -383.369,Z 1181.501,A 0.000,B 0.000,C 90.000,E1 270.115} C_DIS
LIN {X 0.018,Y -375.594,Z 1181.500,A 0.000,B 0.000,C 90.000,E1 270.057} C_DIS
LIN {X 0.124,Y -364.211,Z 1181.500,A 0.000,B 0.000,C 90.000,E1 270.000} C_DIS
LIN {X 0.037,Y -181.562,Z 1181.500,A 0.000,B 0.000,C 90.000,E1 270.000} C_DIS
LIN {X 0.078,Y -180.842,Z 1181.472,A 0.000,B 0.000,C 90.000,E1 264.894} C_DIS
LIN {X -0.019,Y -178.950,Z 1181.444,A 0.000,B 0.000,C 90.000,E1 259.859} C_DIS
LIN {X -0.003,Y -176.854,Z 1181.425,A 0.000,B 0.000,C 90.000,E1 256.464} C_DIS
LIN {X -0.031,Y -175.514,Z 1181.411,A 0.000,B 0.000,C 90.000,E1 253.921} C_DIS
LIN {X 0.031,Y -172.252,Z 1181.387,A 0.000,B 0.000,C 90.000,E1 249.625} C_DIS
LIN {X 0.010,Y -171.730,Z 1181.382,A 0.000,B 0.000,C 90.000,E1 248.773} C_DIS
LIN {X 0.019,Y -167.327,Z 1181.353,A 0.000,B 0.000,C 90.000,E1 243.589} C_DIS
LIN {X -0.049,Y -166.711,Z 1181.349,A 0.000,B 0.000,C 90.000,E1 242.743} C_DIS
LIN {X 0.089,Y -162.691,Z 1181.324,A 0.000,B 0.000,C 90.000,E1 238.329} C_DIS
LIN {X -0.073,Y -161.382,Z 1181.314,A 0.000,B 0.000,C 90.000,E1 236.628} C_DIS
LIN {X -0.029,Y -157.374,Z 1181.290,A 0.000,B 0.000,C 90.000,E1 232.190} C_DIS
LIN {X 0.004,Y -155.368,Z 1181.275,A 0.000,B 0.000,C 90.000,E1 229.504} C_DIS
LIN {X 0.052,Y -151.708,Z 1181.250,A 0.000,B 0.000,C 90.000,E1 225.000} C_DIS
LIN {X 0.062,Y -149.899,Z 1181.235,A 0.000,B 0.000,C 90.000,E1 222.285} C_DIS
LIN {X 0.085,Y -146.758,Z 1181.210,A 0.000,B 0.000,C 90.000,E1 217.729} C_DIS
LIN {X -0.017,Y -145.325,Z 1181.195,A 0.000,B 0.000,C 90.000,E1 215.025} C_DIS
LIN {X 0.023,Y -142.409,Z 1181.164,A 0.000,B 0.000,C 90.000,E1 209.489} C_DIS
LIN {X -0.051,Y -141.393,Z 1181.148,A 0.000,B 0.000,C 90.000,E1 206.744} C_DIS
LIN {X -0.062,Y -139.352,Z 1181.112,A 0.000,B 0.000,C 90.000,E1 200.248} C_DIS
LIN {X 0.058,Y -138.792,Z 1181.097,A 0.000,B 0.000,C 90.000,E1 197.402} C_DIS
LIN {X -0.020,Y -138.346,Z 1181.055,A 0.000,B 0.000,C 90.000,E1 189.962} C_DIS
LIN {X -0.003,Y -139.380,Z 1181.009,A 0.000,B 0.000,C 90.000,E1 181.547} C_DIS
LIN {X 0.051,Y -141.271,Z 1180.972,A 0.000,B 0.000,C 90.000,E1 175.008} C_DIS
LIN {X 0.009,Y -142.637,Z 1180.957,A 0.000,B 0.000,C 90.000,E1 172.243} C_DIS
LIN {X -0.040,Y -144.967,Z 1180.931,A 0.000,B 0.000,C 90.000,E1 167.645} C_DIS
LIN {X -0.049,Y -147.595,Z 1180.911,A 0.000,B 0.000,C 90.000,E1 163.976} C_DIS
LIN {X -0.020,Y -150.212,Z 1180.891,A 0.000,B 0.000,C 90.000,E1 160.315} C_DIS
LIN {X 0.048,Y -153.599,Z 1180.870,A 0.000,B 0.000,C 90.000,E1 156.666} C_DIS
LIN {X 0.035,Y -157.015,Z 1180.850,A 0.000,B 0.000,C 90.000,E1 153.076} C_DIS
LIN {X -0.032,Y -161.134,Z 1180.831,A 0.000,B 0.000,C 90.000,E1 149.537} C_DIS
LIN {X 0.051,Y -163.234,Z 1180.821,A 0.000,B 0.000,C 90.000,E1 147.740} C_DIS
LIN {X -0.083,Y -167.667,Z 1180.801,A 0.000,B 0.000,C 90.000,E1 144.276} C_DIS
LIN {X 0.064,Y -171.490,Z 1180.787,A 0.000,B 0.000,C 90.000,E1 141.618} C_DIS
LIN {X 0.108,Y -176.422,Z 1180.768,A 0.000,B 0.000,C 90.000,E1 138.162} C_DIS
LIN {X -0.020,Y -180.717,Z 1180.754,A 0.000,B 0.000,C 90.000,E1 135.648} C_DIS
LIN {X -0.038,Y -186.121,Z 1180.735,A 0.000,B 0.000,C 90.000,E1 132.285} C_DIS
LIN {X 0.018,Y -190.758,Z 1180.721,A 0.000,B 0.000,C 90.000,E1 129.769} C_DIS
LIN {X -0.073,Y -196.513,Z 1180.703,A 0.000,B 0.000,C 90.000,E1 126.503} C_DIS
LIN {X -0.057,Y -201.184,Z 1180.689,A 0.000,B 0.000,C 90.000,E1 124.119} C_DIS
LIN {X 0.017,Y -201.228,Z 1180.689,A 0.000,B 0.000,C 90.000,E1 124.072} C_DIS
LIN {X -0.021,Y -310.186,Z 1180.689,A 0.000,B 0.000,C 90.000,E1 124.072} C_DIS
LIN {X 0.008,Y -312.471,Z 1180.689,A 0.000,B 0.000,C 90.000,E1 124.040} C_DIS
LIN {X 0.032,Y -315.749,Z 1180.688,A 0.000,B 0.000,C 90.000,E1 123.913} C_DIS
LIN {X -0.123,Y -319.067,Z 1180.687,A 0.000,B 0.000,C 90.000,E1 123.706} C_DIS
LIN {X 0.100,Y -322.732,Z 1180.685,A 0.000,B 0.000,C 90.000,E1 123.245} C_DIS
LIN {X -0.029,Y -324.612,Z 1180.683,A 0.000,B 0.000,C 90.000,E1 122.959} C_DIS
LIN {X 0.112,Y -326.080,Z 1180.681,A 0.000,B 0.000,C 90.000,E1 122.625} C_DIS
LIN {X -0.068,Y -339.417,Z 1180.662,A 0.000,B 0.000,C 90.000,E1 119.205} C_DIS
LIN {X -0.051,Y -351.806,Z 1180.647,A 0.000,B 0.000,C 90.000,E1 116.437} C_DIS
LIN {X 0.177,Y -365.688,Z 1180.632,A 0.000,B 0.000,C 90.000,E1 113.695} C_DIS
LIN {X 0.096,Y -379.384,Z 1180.619,A 0.000,B 0.000,C 90.000,E1 111.354} C_DIS
LIN {X -0.138,Y -394.455,Z 1180.606,A 0.000,B 0.000,C 90.000,E1 109.087} C_DIS
LIN {X 0.116,Y -411.008,Z 1180.593,A 0.000,B 0.000,C 90.000,E1 106.804} C_DIS
LIN {X -0.136,Y -429.159,Z 1180.581,A 0.000,B 0.000,C 90.000,E1 104.647} C_DIS
LIN {X -0.108,Y -448.808,Z 1180.570,A 0.000,B 0.000,C 90.000,E1 102.535} C_DIS
LIN {X -0.207,Y -469.137,Z 1180.559,A 0.000,B 0.000,C 90.000,E1 100.602} C_DIS
LIN {X -0.184,Y -471.468,Z 1180.557,A 0.000,B 0.000,C 90.000,E1 100.366} C_DIS
LIN {X 0.186,Y -473.319,Z 1180.556,A 0.000,B 0.000,C 90.000,E1 100.074} C_DIS
LIN {X 0.010,Y -474.718,Z 1180.555,A 0.000,B 0.000,C 90.000,E1 99.849} C_DIS
LIN {X 0.205,Y -476.544,Z 1180.552,A 0.000,B 0.000,C 90.000,E1 99.321} C_DIS
LIN {X -0.139,Y -477.274,Z 1180.549,A 0.000,B 0.000,C 90.000,E1 98.859} C_DIS
LIN {X 0.000,Y -477.031,Z 1180.546,A 0.000,B 0.000,C 90.000,E1 98.341} C_DIS
LIN {X 0.211,Y -475.782,Z 1180.544,A 0.000,B 0.000,C 90.000,E1 97.814} C_DIS
LIN {X 0.015,Y -474.720,Z 1180.542,A 0.000,B 0.000,C 90.000,E1 97.587} C_DIS
LIN {X -0.118,Y -473.296,Z 1180.541,A 0.000,B 0.000,C 90.000,E1 97.352} C_DIS
LIN {X -0.184,Y -458.827,Z 1180.530,A 0.000,B 0.000,C 90.000,E1 95.334} C_DIS
LIN {X -0.056,Y -439.497,Z 1180.514,A 0.000,B 0.000,C 90.000,E1 92.465} C_DIS
LIN {X 0.180,Y -423.321,Z 1180.499,A 0.000,B 0.000,C 90.000,E1 89.771} C_DIS
LIN {X -0.123,Y -410.009,Z 1180.485,A 0.000,B 0.000,C 90.000,E1 87.364} C_DIS
LIN {X -0.035,Y -399.704,Z 1180.474,A 0.000,B 0.000,C 90.000,E1 85.412} C_DIS
LIN {X -0.085,Y -387.939,Z 1180.462,A 0.000,B 0.000,C 90.000,E1 83.166} C_DIS
LIN {X 0.028,Y -379.168,Z 1180.452,A 0.000,B 0.000,C 90.000,E1 81.432} C_DIS
LIN {X 0.036,Y -370.130,Z 1180.443,A 0.000,B 0.000,C 90.000,E1 79.690} C_DIS
LIN {X -0.052,Y -360.779,Z 1180.433,A 0.000,B 0.000,C 90.000,E1 77.937} C_DIS
LIN {X 0.057,Y -349.591,Z 1180.421,A 0.000,B 0.000,C 90.000,E1 75.825} C_DIS
LIN {X 0.086,Y -338.289,Z 1180.409,A 0.000,B 0.000,C 90.000,E1 73.685} C_DIS
LIN {X -0.061,Y -325.587,Z 1180.396,A 0.000,B 0.000,C 90.000,E1 71.221} C_DIS
LIN {X -0.034,Y -310.458,Z 1180.378,A 0.000,B 0.000,C 90.000,E1 68.028} C_DIS
LIN {X 0.048,Y -294.926,Z 1180.358,A 0.000,B 0.000,C 90.000,E1 64.409} C_DIS
LIN {X 0.074,Y -284.347,Z 1180.343,A 0.000,B 0.000,C 90.000,E1 61.719} C_DIS
LIN {X -0.057,Y -273.086,Z 1180.326,A 0.000,B 0.000,C 90.000,E1 58.663} C_DIS
LIN {X -0.116,Y -263.518,Z 1180.310,A 0.000,B 0.000,C 90.000,E1 55.881} C_DIS
LIN {X 0.085,Y -252.170,Z 1180.291,A 0.000,B 0.000,C 90.000,E1 52.271} C_DIS
LIN {X 0.021,Y -242.618,Z 1180.272,A 0.000,B 0.000,C 90.000,E1 49.013} C_DIS
LIN {X -0.049,Y -232.676,Z 1180.252,A 0.000,B 0.000,C 90.000,E1 45.324} C_DIS
LIN {X 0.066,Y -223.712,Z 1180.231,A 0.000,B 0.000,C 90.000,E1 41.515} C_DIS
LIN {X -0.012,Y -215.533,Z 1180.209,A 0.000,B 0.000,C 90.000,E1 37.684} C_DIS
LIN {X -0.076,Y -208.180,Z 1180.188,A 0.000,B 0.000,C 90.000,E1 33.785} C_DIS
LIN {X -0.028,Y -201.543,Z 1180.166,A 0.000,B 0.000,C 90.000,E1 29.795} C_DIS
LIN {X 0.111,Y -195.619,Z 1180.143,A 0.000,B 0.000,C 90.000,E1 25.720} C_DIS
LIN {X 0.009,Y -190.544,Z 1180.120,A 0.000,B 0.000,C 90.000,E1 21.663} C_DIS
LIN {X 0.074,Y -186.329,Z 1180.097,A 0.000,B 0.000,C 90.000,E1 17.511} C_DIS
LIN {X -0.024,Y -182.636,Z 1180.070,A 0.000,B 0.000,C 90.000,E1 12.535} C_DIS
LIN {X -0.077,Y -180.050,Z 1180.037,A 0.000,B 0.000,C 90.000,E1 6.663} C_DIS
LIN {X -0.082,Y -181.206,Z 1179.969,A 0.000,B 0.000,C 90.000,E1 354.489} C_DIS
LIN {X 0.060,Y -184.174,Z 1179.941,A 0.000,B 0.000,C 90.000,E1 349.398} C_DIS
LIN {X 0.040,Y -187.734,Z 1179.918,A 0.000,B 0.000,C 90.000,E1 345.227} C_DIS
LIN {X 0.013,Y -192.222,Z 1179.895,A 0.000,B 0.000,C 90.000,E1 341.094} C_DIS
LIN {X 0.009,Y -197.449,Z 1179.872,A 0.000,B 0.000,C 90.000,E1 336.997} C_DIS
LIN {X 0.003,Y -203.293,Z 1179.850,A 0.000,B 0.000,C 90.000,E1 332.948} C_DIS
LIN {X 0.015,Y -209.865,Z 1179.828,A 0.000,B 0.000,C 90.000,E1 328.948} C_DIS
LIN {X -0.038,Y -216.968,Z 1179.806,A 0.000,B 0.000,C 90.000,E1 325.022} C_DIS
LIN {X -0.001,Y -223.161,Z 1179.788,A 0.000,B 0.000,C 90.000,E1 321.904} C_DIS
LIN {X -0.064,Y -230.317,Z 1179.771,A 0.000,B 0.000,C 90.000,E1 318.852} C_DIS
LIN {X -0.003,Y -239.689,Z 1179.752,A 0.000,B 0.000,C 90.000,E1 315.445} C_DIS
LIN {X -0.005,Y -250.458,Z 1179.734,A 0.000,B 0.000,C 90.000,E1 312.123} C_DIS
LIN {X -0.004,Y -262.569,Z 1179.716,A 0.000,B 0.000,C 90.000,E1 308.874} C_DIS
LIN {X 0.106,Y -272.825,Z 1179.702,A 0.000,B 0.000,C 90.000,E1 306.377} C_DIS
LIN {X -0.083,Y -284.198,Z 1179.689,A 0.000,B 0.000,C 90.000,E1 303.992} C_DIS
LIN {X 0.052,Y -296.977,Z 1179.676,A 0.000,B 0.000,C 90.000,E1 301.592} C_DIS
LIN {X 0.060,Y -313.000,Z 1179.661,A 0.000,B 0.000,C 90.000,E1 298.949} C_DIS
LIN {X 0.144,Y -321.729,Z 1179.654,A 0.000,B 0.000,C 90.000,E1 297.641} C_DIS
LIN {X -0.105,Y -331.211,Z 1179.647,A 0.000,B 0.000,C 90.000,E1 296.411} C_DIS
LIN {X 0.009,Y -344.019,Z 1179.638,A 0.000,B 0.000,C 90.000,E1 294.847} C_DIS
LIN {X 0.041,Y -362.776,Z 1179.627,A 0.000,B 0.000,C 90.000,E1 292.770} C_DIS
LIN {X -0.006,Y -389.990,Z 1179.612,A 0.000,B 0.000,C 90.000,E1 290.120} C_DIS
LIN {X -0.023,Y -400.430,Z 1179.606,A 0.000,B 0.000,C 90.000,E1 289.141} C_DIS
LIN {X 0.111,Y -408.394,Z 1179.602,A 0.000,B 0.000,C 90.000,E1 288.362} C_DIS
LIN {X 0.108,Y -418.604,Z 1179.596,A 0.000,B 0.000,C 90.000,E1 287.330} C_DIS
LIN {X -0.035,Y -426.055,Z 1179.592,A 0.000,B 0.000,C 90.000,E1 286.551} C_DIS
LIN {X 0.062,Y -435.417,Z 1179.586,A 0.000,B 0.000,C 90.000,E1 285.481} C_DIS
LIN {X -0.191,Y -441.837,Z 1179.582,A 0.000,B 0.000,C 90.000,E1 284.717} C_DIS
LIN {X -0.086,Y -445.759,Z 1179.579,A 0.000,B 0.000,C 90.000,E1 284.175} C_DIS
LIN {X 0.169,Y -450.984,Z 1179.574,A 0.000,B 0.000,C 90.000,E1 283.355} C_DIS
LIN {X 0.040,Y -455.598,Z 1179.570,A 0.000,B 0.000,C 90.000,E1 282.591} C_DIS
LIN {X -0.053,Y -459.557,Z 1179.566,A 0.000,B 0.000,C 90.000,E1 281.827} C_DIS
LIN {X 0.055,Y -461.834,Z 1179.563,A 0.000,B 0.000,C 90.000,E1 281.299} C_DIS
LIN {X 0.089,Y -463.842,Z 1179.560,A 0.000,B 0.000,C 90.000,E1 280.782} C_DIS
LIN {X -0.183,Y -467.240,Z 1179.554,A 0.000,B 0.000,C 90.000,E1 279.792} C_DIS
LIN {X 0.048,Y -469.837,Z 1179.549,A 0.000,B 0.000,C 90.000,E1 278.746} C_DIS
LIN {X 0.209,Y -470.847,Z 1179.546,A 0.000,B 0.000,C 90.000,E1 278.219} C_DIS
LIN {X -0.158,Y -471.476,Z 1179.543,A 0.000,B 0.000,C 90.000,E1 277.757} C_DIS
LIN {X -0.051,Y -471.729,Z 1179.540,A 0.000,B 0.000,C 90.000,E1 277.239} C_DIS
LIN {X 0.060,Y -471.608,Z 1179.537,A 0.000,B 0.000,C 90.000,E1 276.720} C_DIS
LIN {X 0.173,Y -471.004,Z 1179.535,A 0.000,B 0.000,C 90.000,E1 276.201} C_DIS
LIN {X -0.183,Y -469.963,Z 1179.532,A 0.000,B 0.000,C 90.000,E1 275.739} C_DIS
LIN {X -0.076,Y -468.522,Z 1179.529,A 0.000,B 0.000,C 90.000,E1 275.220} C_DIS
LIN {X -0.181,Y -465.516,Z 1179.525,A 0.000,B 0.000,C 90.000,E1 274.473} C_DIS
LIN {X -0.101,Y -462.804,Z 1179.522,A 0.000,B 0.000,C 90.000,E1 273.955} C_DIS
LIN {X -0.067,Y -459.362,Z 1179.519,A 0.000,B 0.000,C 90.000,E1 273.440} C_DIS
LIN {X -0.023,Y -454.946,Z 1179.516,A 0.000,B 0.000,C 90.000,E1 272.922} C_DIS
LIN {X 0.206,Y -452.284,Z 1179.515,A 0.000,B 0.000,C 90.000,E1 272.636} C_DIS
LIN {X -0.051,Y -446.236,Z 1179.512,A 0.000,B 0.000,C 90.000,E1 272.178} C_DIS
LIN {X 0.209,Y -439.449,Z 1179.510,A 0.000,B 0.000,C 90.000,E1 271.718} C_DIS
LIN {X 0.193,Y -432.488,Z 1179.508,A 0.000,B 0.000,C 90.000,E1 271.375} C_DIS
LIN {X -0.195,Y -425.554,Z 1179.506,A 0.000,B 0.000,C 90.000,E1 271.146} C_DIS
LIN {X -0.165,Y -415.261,Z 1179.504,A 0.000,B 0.000,C 90.000,E1 270.802} C_DIS
LIN {X -0.078,Y -404.675,Z 1179.503,A 0.000,B 0.000,C 90.000,E1 270.516} C_DIS
LIN {X 0.019,Y -394.036,Z 1179.502,A 0.000,B 0.000,C 90.000,E1 270.286} C_DIS
LIN {X -0.048,Y -382.509,Z 1179.501,A 0.000,B 0.000,C 90.000,E1 270.115} C_DIS
LIN {X -0.153,Y -374.025,Z 1179.500,A 0.000,B 0.000,C 90.000,E1 270.057} C_DIS
LIN {X 0.060,Y -367.867,Z 1179.500,A 0.000,B 0.000,C 90.000,E1 270.000} C_DIS
LIN {X 0.007,Y -181.561,Z 1179.500,A 0.000,B 0.000,C 90.000,E1 270.000} C_DIS
LIN {X 0.015,Y -180.835,Z 1179.472,A 0.000,B 0.000,C 90.000,E1 264.894} C_DIS
LIN {X 0.094,Y -178.943,Z 1179.443,A 0.000,B 0.000,C 90.000,E1 259.803} C_DIS
LIN {X -0.038,Y -175.993,Z 1179.415,A 0.000,B 0.000,C 90.000,E1 254.755} C_DIS
LIN {X -0.093,Y -175.497,Z 1179.411,A 0.000,B 0.000,C 90.000,E1 253.921} C_DIS
LIN {X -0.030,Y -172.240,Z 1179.387,A 0.000,B 0.000,C 90.000,E1 249.625} C_DIS
LIN {X -0.051,Y -171.717,Z 1179.382,A 0.000,B 0.000,C 90.000,E1 248.773} C_DIS
LIN {X -0.040,Y -167.312,Z 1179.353,A 0.000,B 0.000,C 90.000,E1 243.589} C_DIS
LIN {X 0.040,Y -166.694,Z 1179.348,A 0.000,B 0.000,C 90.000,E1 242.692} C_DIS
LIN {X 0.030,Y -162.675,Z 1179.324,A 0.000,B 0.000,C 90.000,E1 238.329} C_DIS
LIN {X 0.003,Y -161.365,Z 1179.314,A 0.000,B 0.000,C 90.000,E1 236.580} C_DIS
LIN {X -0.088,Y -157.358,Z 1179.290,A 0.000,B 0.000,C 90.000,E1 232.190} C_DIS
LIN {X 0.065,Y -155.347,Z 1179.275,A 0.000,B 0.000,C 90.000,E1 229.461} C_DIS
LIN {X -0.005,Y -151.693,Z 1179.250,A 0.000,B 0.000,C 90.000,E1 225.000} C_DIS
LIN {X 0.043,Y -150.555,Z 1179.240,A 0.000,B 0.000,C 90.000,E1 223.176} C_DIS
LIN {X -0.040,Y -147.282,Z 1179.215,A 0.000,B 0.000,C 90.000,E1 218.669} C_DIS
LIN {X -0.072,Y -145.311,Z 1179.194,A 0.000,B 0.000,C 90.000,E1 215.025} C_DIS
LIN {X 0.039,Y -142.400,Z 1179.164,A 0.000,B 0.000,C 90.000,E1 209.461} C_DIS
LIN {X 0.021,Y -141.383,Z 1179.148,A 0.000,B 0.000,C 90.000,E1 206.693} C_DIS
LIN {X 0.014,Y -139.350,Z 1179.112,A 0.000,B 0.000,C 90.000,E1 200.194} C_DIS
LIN {X 0.004,Y -138.786,Z 1179.097,A 0.000,B 0.000,C 90.000,E1 197.402} C_DIS
LIN {X 0.062,Y -138.345,Z 1179.055,A 0.000,B 0.000,C 90.000,E1 189.905} C_DIS
LIN {X -0.056,Y -139.385,Z 1179.008,A 0.000,B 0.000,C 90.000,E1 181.547} C_DIS
LIN {X -0.003,Y -141.281,Z 1178.972,A 0.000,B 0.000,C 90.000,E1 175.008} C_DIS
LIN {X -0.045,Y -142.646,Z 1178.957,A 0.000,B 0.000,C 90.000,E1 172.243} C_DIS
LIN {X 0.046,Y -144.981,Z 1178.931,A 0.000,B 0.000,C 90.000,E1 167.589} C_DIS
LIN {X 0.037,Y -147.608,Z 1178.911,A 0.000,B 0.000,C 90.000,E1 163.921} C_DIS
LIN {X -0.026,Y -150.230,Z 1178.891,A 0.000,B 0.000,C 90.000,E1 160.296} C_DIS
LIN {X -0.010,Y -153.620,Z 1178.870,A 0.000,B 0.000,C 90.000,E1 156.666} C_DIS
LIN {X -0.023,Y -157.036,Z 1178.850,A 0.000,B 0.000,C 90.000,E1 153.076} C_DIS
LIN {X -0.092,Y -161.161,Z 1178.831,A 0.000,B 0.000,C 90.000,E1 149.537} C_DIS
LIN {X -0.009,Y -163.258,Z 1178.821,A 0.000,B 0.000,C 90.000,E1 147.740} C_DIS
LIN {X 0.090,Y -167.696,Z 1178.801,A 0.000,B 0.000,C 90.000,E1 144.196} C_DIS
LIN {X 0.003,Y -171.517,Z 1178.787,A 0.000,B 0.000,C 90.000,E1 141.618} C_DIS
LIN {X 0.047,Y -176.454,Z 1178.768,A 0.000,B 0.000,C 90.000,E1 138.162} C_DIS
LIN {X -0.083,Y -180.751,Z 1178.753,A 0.000,B 0.000,C 90.000,E1 135.648} C_DIS
LIN {X 0.034,Y -186.155,Z 1178.735,A 0.000,B 0.000,C 90.000,E1 132.243} C_DIS
LIN {X -0.047,Y -190.793,Z 1178.721,A 0.000,B 0.000,C 90.000,E1 129.769} C_DIS
LIN {X 0.018,Y -196.550,Z 1178.703,A 0.000,B 0.000,C 90.000,E1 126.457} C_DIS
LIN {X -0.019,Y -201.166,Z 1178.690,A 0.000,B 0.000,C 90.000,E1 124.119} C_DIS
LIN {X 0.056,Y -201.210,Z 1178.689,A 0.000,B 0.000,C 90.000,E1 124.072} C_DIS
LIN {X 0.051,Y -310.996,Z 1178.689,A 0.000,B 0.000,C 90.000,E1 124.072} C_DIS
LIN {X -0.097,Y -313.711,Z 1178.689,A 0.000,B 0.000,C 90.000,E1 124.040} C_DIS
LIN {X 0.066,Y -317.166,Z 1178.688,A 0.000,B 0.000,C 90.000,E1 123.833} C_DIS
LIN {X 0.173,Y -320.691,Z 1178.686,A 0.000,B 0.000,C 90.000,E1 123.499} C_DIS
LIN {X -0.111,Y -324.274,Z 1178.683,A 0.000,B 0.000,C 90.000,E1 123.038} C_DIS
LIN {X 0.151,Y -325.837,Z 1178.682,A 0.000,B 0.000,C 90.000,E1 122.673} C_DIS
LIN {X -0.057,Y -339.179,Z 1178.662,A 0.000,B 0.000,C 90.000,E1 119.255} C_DIS
LIN {X -0.051,Y -351.538,Z 1178.647,A 0.000,B 0.000,C 90.000,E1 116.488} C_DIS
LIN {X 0.010,Y -365.394,Z 1178.632,A 0.000,B 0.000,C 90.000,E1 113.770} C_DIS
LIN {X 0.062,Y -379.063,Z 1178.619,A 0.000,B 0.000,C 90.000,E1 111.408} C_DIS
LIN {X 0.185,Y -394.105,Z 1178.606,A 0.000,B 0.000,C 90.000,E1 109.087} C_DIS
LIN {X 0.051,Y -410.625,Z 1178.594,A 0.000,B 0.000,C 90.000,E1 106.858} C_DIS
LIN {X 0.088,Y -428.742,Z 1178.582,A 0.000,B 0.000,C 90.000,E1 104.662} C_DIS
LIN {X 0.207,Y -448.383,Z 1178.570,A 0.000,B 0.000,C 90.000,E1 102.535} C_DIS
LIN {X 0.135,Y -471.083,Z 1178.558,A 0.000,B 0.000,C 90.000,E1 100.366} C_DIS
LIN {X 0.092,Y -472.897,Z 1178.556,A 0.000,B 0.000,C 90.000,E1 100.141} C_DIS
LIN {X -0.049,Y -474.404,Z 1178.555,A 0.000,B 0.000,C 90.000,E1 99.905} C_DIS
LIN {X -0.192,Y -475.531,Z 1178.554,A 0.000,B 0.000,C 90.000,E1 99.670} C_DIS
LIN {X -0.070,Y -476.875,Z 1178.551,A 0.000,B 0.000,C 90.000,E1 99.151} C_DIS
LIN {X 0.135,Y -477.197,Z 1178.548,A 0.000,B 0.000,C 90.000,E1 98.624} C_DIS
LIN {X -0.196,Y -476.551,Z 1178.545,A 0.000,B 0.000,C 90.000,E1 98.163} C_DIS
LIN {X -0.052,Y -474.835,Z 1178.542,A 0.000,B 0.000,C 90.000,E1 97.644} C_DIS
LIN {X -0.186,Y -473.480,Z 1178.541,A 0.000,B 0.000,C 90.000,E1 97.409} C_DIS
LIN {X 0.210,Y -459.050,Z 1178.530,A 0.000,B 0.000,C 90.000,E1 95.334} C_DIS
LIN {X -0.106,Y -439.736,Z 1178.514,A 0.000,B 0.000,C 90.000,E1 92.522} C_DIS
LIN {X -0.162,Y -422.012,Z 1178.498,A 0.000,B 0.000,C 90.000,E1 89.599} C_DIS
LIN {X -0.081,Y -408.713,Z 1178.484,A 0.000,B 0.000,C 90.000,E1 87.135} C_DIS
LIN {X 0.008,Y -398.404,Z 1178.473,A 0.000,B 0.000,C 90.000,E1 85.179} C_DIS
LIN {X -0.063,Y -386.647,Z 1178.461,A 0.000,B 0.000,C 90.000,E1 82.932} C_DIS
LIN {X 0.031,Y -377.842,Z 1178.451,A 0.000,B 0.000,C 90.000,E1 81.197} C_DIS
LIN {X 0.019,Y -368.747,Z 1178.441,A 0.000,B 0.000,C 90.000,E1 79.454} C_DIS
LIN {X -0.091,Y -359.364,Z 1178.432,A 0.000,B 0.000,C 90.000,E1 77.701} C_DIS
LIN {X -0.012,Y -348.154,Z 1178.420,A 0.000,B 0.000,C 90.000,E1 75.589} C_DIS
LIN {X -0.012,Y -336.829,Z 1178.408,A 0.000,B 0.000,C 90.000,E1 73.449} C_DIS
LIN {X 0.179,Y -322.624,Z 1178.392,A 0.000,B 0.000,C 90.000,E1 70.604} C_DIS
LIN {X 0.077,Y -309.131,Z 1178.376,A 0.000,B 0.000,C 90.000,E1 67.741} C_DIS
LIN {X 0.079,Y -295.048,Z 1178.358,A 0.000,B 0.000,C 90.000,E1 64.460} C_DIS
LIN {X 0.112,Y -284.436,Z 1178.343,A 0.000,B 0.000,C 90.000,E1 61.769} C_DIS
LIN {X -0.150,Y -273.159,Z 1178.326,A 0.000,B 0.000,C 90.000,E1 58.742} C_DIS
LIN {X -0.058,Y -263.556,Z 1178.311,A 0.000,B 0.000,C 90.000,E1 55.928} C_DIS
LIN {X -0.005,Y -252.179,Z 1178.291,A 0.000,B 0.000,C 90.000,E1 52.351} C_DIS
LIN {X 0.090,Y -241.562,Z 1178.271,A 0.000,B 0.000,C 90.000,E1 48.690} C_DIS
LIN {X -0.010,Y -231.712,Z 1178.250,A 0.000,B 0.000,C 90.000,E1 45.000} C_DIS
LIN {X -0.076,Y -222.826,Z 1178.229,A 0.000,B 0.000,C 90.000,E1 41.229} C_DIS
LIN {X -0.040,Y -214.707,Z 1178.208,A 0.000,B 0.000,C 90.000,E1 37.363} C_DIS
LIN {X 0.031,Y -207.377,Z 1178.186,A 0.000,B 0.000,C 90.000,E1 33.420} C_DIS
LIN {X -0.058,Y -200.766,Z 1178.164,A 0.000,B 0.000,C 90.000,E1 29.461} C_DIS
LIN {X -0.031,Y -194.884,Z 1178.141,A 0.000,B 0.000,C 90.000,E1 25.412} C_DIS
LIN {X 0.097,Y -189.885,Z 1178.118,A 0.000,B 0.000,C 90.000,E1 21.280} C_DIS
LIN {X 0.019,Y -185.729,Z 1178.095,A 0.000,B 0.000,C 90.000,E1 17.166} C_DIS
LIN {X -0.034,Y -182.625,Z 1178.072,A 0.000,B 0.000,C 90.000,E1 13.008} C_DIS
LIN {X -0.055,Y -179.861,Z 1178.039,A 0.000,B 0.000,C 90.000,E1 7.125} C_DIS
LIN {X 0.086,Y -180.874,Z 1177.969,A 0.000,B 0.000,C 90.000,E1 354.432} C_DIS
LIN {X 0.035,Y -183.840,Z 1177.941,A 0.000,B 0.000,C 90.000,E1 349.398} C_DIS
LIN {X 0.004,Y -187.387,Z 1177.918,A 0.000,B 0.000,C 90.000,E1 345.227} C_DIS
LIN {X -0.034,Y -191.860,Z 1177.895,A 0.000,B 0.000,C 90.000,E1 341.094} C_DIS
LIN {X 0.025,Y -197.073,Z 1177.872,A 0.000,B 0.000,C 90.000,E1 336.975} C_DIS
LIN {X 0.022,Y -202.949,Z 1177.850,A 0.000,B 0.000,C 90.000,E1 332.922} C_DIS
LIN {X -0.072,Y -209.518,Z 1177.827,A 0.000,B 0.000,C 90.000,E1 328.948} C_DIS
LIN {X 0.038,Y -216.615,Z 1177.805,A 0.000,B 0.000,C 90.000,E1 324.975} C_DIS
LIN {X -0.114,Y -222.879,Z 1177.788,A 0.000,B 0.000,C 90.000,E1 321.904} C_DIS
LIN {X 0.137,Y -230.093,Z 1177.771,A 0.000,B 0.000,C 90.000,E1 318.771} C_DIS
LIN {X 0.037,Y -239.526,Z 1177.752,A 0.000,B 0.000,C 90.000,E1 315.405} C_DIS
LIN {X 0.042,Y -250.346,Z 1177.734,A 0.000,B 0.000,C 90.000,E1 312.081} C_DIS
LIN {X 0.053,Y -262.506,Z 1177.716,A 0.000,B 0.000,C 90.000,E1 308.830} C_DIS
LIN {X -0.048,Y -272.821,Z 1177.702,A 0.000,B 0.000,C 90.000,E1 306.377} C_DIS
LIN {X 0.151,Y -284.238,Z 1177.689,A 0.000,B 0.000,C 90.000,E1 303.913} C_DIS
LIN {X -0.116,Y -297.063,Z 1177.675,A 0.000,B 0.000,C 90.000,E1 301.592} C_DIS
LIN {X -0.115,Y -313.114,Z 1177.661,A 0.000,B 0.000,C 90.000,E1 298.949} C_DIS
LIN {X -0.034,Y -321.846,Z 1177.654,A 0.000,B 0.000,C 90.000,E1 297.641} C_DIS
LIN {X -0.029,Y -333.813,Z 1177.645,A 0.000,B 0.000,C 90.000,E1 296.052} C_DIS
LIN {X -0.176,Y -354.744,Z 1177.631,A 0.000,B 0.000,C 90.000,E1 293.643} C_DIS
LIN {X -0.048,Y -373.626,Z 1177.620,A 0.000,B 0.000,C 90.000,E1 291.663} C_DIS
LIN {X -0.061,Y -392.501,Z 1177.610,A 0.000,B 0.000,C 90.000,E1 289.885} C_DIS
LIN {X 0.237,Y -405.685,Z 1177.604,A 0.000,B 0.000,C 90.000,E1 288.598} C_DIS
LIN {X 0.010,Y -413.343,Z 1177.599,A 0.000,B 0.000,C 90.000,E1 287.873} C_DIS
LIN {X -0.015,Y -420.919,Z 1177.595,A 0.000,B 0.000,C 90.000,E1 287.094} C_DIS
LIN {X 0.212,Y -428.352,Z 1177.590,A 0.000,B 0.000,C 90.000,E1 286.260} C_DIS
LIN {X 0.189,Y -435.249,Z 1177.586,A 0.000,B 0.000,C 90.000,E1 285.481} C_DIS
LIN {X -0.076,Y -441.740,Z 1177.582,A 0.000,B 0.000,C 90.000,E1 284.717} C_DIS
LIN {X 0.250,Y -447.447,Z 1177.577,A 0.000,B 0.000,C 90.000,E1 283.883} C_DIS
LIN {X 0.092,Y -452.500,Z 1177.573,A 0.000,B 0.000,C 90.000,E1 283.119} C_DIS
LIN {X -0.028,Y -456.947,Z 1177.569,A 0.000,B 0.000,C 90.000,E1 282.355} C_DIS
LIN {X -0.108,Y -460.742,Z 1177.564,A 0.000,B 0.000,C 90.000,E1 281.591} C_DIS
LIN {X -0.250,Y -463.888,Z 1177.560,A 0.000,B 0.000,C 90.000,E1 280.838} C_DIS
LIN {X -0.123,Y -465.716,Z 1177.557,A 0.000,B 0.000,C 90.000,E1 280.310} C_DIS
LIN {X -0.064,Y -467.351,Z 1177.554,A 0.000,B 0.000,C 90.000,E1 279.792} C_DIS
LIN {X 0.168,Y -470.018,Z 1177.549,A 0.000,B 0.000,C 90.000,E1 278.746} C_DIS
LIN {X -0.135,Y -471.008,Z 1177.546,A 0.000,B 0.000,C 90.000,E1 278.276} C_DIS
LIN {X -0.036,Y -471.674,Z 1177.543,A 0.000,B 0.000,C 90.000,E1 277.757} C_DIS
LIN {X 0.072,Y -471.984,Z 1177.540,A 0.000,B 0.000,C 90.000,E1 277.239} C_DIS
LIN {X 0.184,Y -471.843,Z 1177.537,A 0.000,B 0.000,C 90.000,E1 276.720} C_DIS
LIN {X -0.169,Y -471.285,Z 1177.535,A 0.000,B 0.000,C 90.000,E1 276.258} C_DIS
LIN {X -0.056,Y -470.275,Z 1177.532,A 0.000,B 0.000,C 90.000,E1 275.739} C_DIS
LIN {X 0.053,Y -468.851,Z 1177.529,A 0.000,B 0.000,C 90.000,E1 275.220} C_DIS
LIN {X 0.153,Y -466.989,Z 1177.526,A 0.000,B 0.000,C 90.000,E1 274.702} C_DIS
LIN {X 0.209,Y -464.624,Z 1177.523,A 0.000,B 0.000,C 90.000,E1 274.188} C_DIS
LIN {X -0.179,Y -461.587,Z 1177.521,A 0.000,B 0.000,C 90.000,E1 273.726} C_DIS
LIN {X 0.066,Y -459.802,Z 1177.519,A 0.000,B 0.000,C 90.000,E1 273.440} C_DIS
LIN {X 0.110,Y -455.441,Z 1177.516,A 0.000,B 0.000,C 90.000,E1 272.922} C_DIS
LIN {X -0.112,Y -452.843,Z 1177.515,A 0.000,B 0.000,C 90.000,E1 272.694} C_DIS
LIN {X 0.182,Y -449.999,Z 1177.514,A 0.000,B 0.000,C 90.000,E1 272.407} C_DIS
LIN {X 0.026,Y -446.783,Z 1177.512,A 0.000,B 0.000,C 90.000,E1 272.178} C_DIS
LIN {X -0.134,Y -440.176,Z 1177.510,A 0.000,B 0.000,C 90.000,E1 271.776} C_DIS
LIN {X -0.186,Y -433.252,Z 1177.508,A 0.000,B 0.000,C 90.000,E1 271.432} C_DIS
LIN {X -0.197,Y -426.271,Z 1177.506,A 0.000,B 0.000,C 90.000,E1 271.146} C_DIS
LIN {X 0.121,Y -419.241,Z 1177.505,A 0.000,B 0.000,C 90.000,E1 270.859} C_DIS
LIN {X 0.030,Y -408.596,Z 1177.503,A 0.000,B 0.000,C 90.000,E1 270.573} C_DIS
LIN {X -0.022,Y -397.590,Z 1177.502,A 0.000,B 0.000,C 90.000,E1 270.344} C_DIS
LIN {X -0.127,Y -386.907,Z 1177.501,A 0.000,B 0.000,C 90.000,E1 270.172} C_DIS
LIN {X -0.094,Y -377.520,Z 1177.500,A 0.000,B 0.000,C 90.000,E1 270.057} C_DIS
LIN {X -0.040,Y -368.006,Z 1177.500,A 0.000,B 0.000,C 90.000,E1 270.000} C_DIS
LIN {X -0.043,Y -181.559,Z 1177.500,A 0.000,B 0.000,C 90.000,E1 270.000} C_DIS
LIN {X -0.036,Y -180.831,Z 1177.472,A 0.000,B 0.000,C 90.000,E1 264.894} C_DIS
LIN {X 0.043,Y -178.937,Z 1177.443,A 0.000,B 0.000,C 90.000,E1 259.803} C_DIS
LIN {X -0.089,Y -175.986,Z 1177.415,A 0.000,B 0.000,C 90.000,E1 254.755} C_DIS
LIN {X 0.026,Y -175.484,Z 1177.410,A 0.000,B 0.000,C 90.000,E1 253.866} C_DIS
LIN {X 0.082,Y -172.229,Z 1177.387,A 0.000,B 0.000,C 90.000,E1 249.571} C_DIS
LIN {X 0.060,Y -171.706,Z 1177.382,A 0.000,B 0.000,C 90.000,E1 248.720} C_DIS
LIN {X -0.015,Y -167.301,Z 1177.353,A 0.000,B 0.000,C 90.000,E1 243.563} C_DIS
LIN {X -0.009,Y -166.680,Z 1177.348,A 0.000,B 0.000,C 90.000,E1 242.692} C_DIS
LIN {X -0.018,Y -162.662,Z 1177.324,A 0.000,B 0.000,C 90.000,E1 238.329} C_DIS
LIN {X -0.045,Y -161.351,Z 1177.314,A 0.000,B 0.000,C 90.000,E1 236.580} C_DIS
LIN {X -0.010,Y -157.345,Z 1177.290,A 0.000,B 0.000,C 90.000,E1 232.145} C_DIS
LIN {X 0.019,Y -155.331,Z 1177.275,A 0.000,B 0.000,C 90.000,E1 229.461} C_DIS
LIN {X -0.051,Y -151.681,Z 1177.250,A 0.000,B 0.000,C 90.000,E1 225.000} C_DIS
LIN {X -0.003,Y -150.545,Z 1177.240,A 0.000,B 0.000,C 90.000,E1 223.176} C_DIS
LIN {X 0.029,Y -147.272,Z 1177.215,A 0.000,B 0.000,C 90.000,E1 218.624} C_DIS
LIN {X 0.002,Y -145.299,Z 1177.194,A 0.000,B 0.000,C 90.000,E1 214.978} C_DIS
LIN {X -0.006,Y -142.394,Z 1177.164,A 0.000,B 0.000,C 90.000,E1 209.461} C_DIS
LIN {X -0.022,Y -141.374,Z 1177.148,A 0.000,B 0.000,C 90.000,E1 206.693} C_DIS
LIN {X 0.019,Y -139.346,Z 1177.112,A 0.000,B 0.000,C 90.000,E1 200.174} C_DIS
LIN {X -0.039,Y -138.782,Z 1177.097,A 0.000,B 0.000,C 90.000,E1 197.402} C_DIS
LIN {X 0.019,Y -138.343,Z 1177.055,A 0.000,B 0.000,C 90.000,E1 189.905} C_DIS
LIN {X 0.039,Y -139.391,Z 1177.008,A 0.000,B 0.000,C 90.000,E1 181.489} C_DIS
LIN {X -0.047,Y -141.289,Z 1176.972,A 0.000,B 0.000,C 90.000,E1 175.008} C_DIS
LIN {X 0.052,Y -142.653,Z 1176.957,A 0.000,B 0.000,C 90.000,E1 172.186} C_DIS
LIN {X 0.002,Y -144.992,Z 1176.931,A 0.000,B 0.000,C 90.000,E1 167.589} C_DIS
LIN {X -0.009,Y -147.619,Z 1176.911,A 0.000,B 0.000,C 90.000,E1 163.921} C_DIS
LIN {X 0.070,Y -150.244,Z 1176.890,A 0.000,B 0.000,C 90.000,E1 160.242} C_DIS
LIN {X -0.056,Y -153.639,Z 1176.870,A 0.000,B 0.000,C 90.000,E1 156.666} C_DIS
LIN {X 0.001,Y -157.055,Z 1176.850,A 0.000,B 0.000,C 90.000,E1 153.050} C_DIS
LIN {X 0.000,Y -161.183,Z 1176.830,A 0.000,B 0.000,C 90.000,E1 149.488} C_DIS
LIN {X 0.030,Y -163.276,Z 1176.821,A 0.000,B 0.000,C 90.000,E1 147.709} C_DIS
LIN {X 0.040,Y -167.720,Z 1176.801,A 0.000,B 0.000,C 90.000,E1 144.196} C_DIS
LIN {X -0.047,Y -171.538,Z 1176.787,A 0.000,B 0.000,C 90.000,E1 141.618} C_DIS
LIN {X -0.004,Y -176.479,Z 1176.768,A 0.000,B 0.000,C 90.000,E1 138.162} C_DIS
LIN {X -0.005,Y -180.777,Z 1176.753,A 0.000,B 0.000,C 90.000,E1 135.607} C_DIS
LIN {X -0.018,Y -186.183,Z 1176.735,A 0.000,B 0.000,C 90.000,E1 132.243} C_DIS
LIN {X 0.047,Y -190.821,Z 1176.721,A 0.000,B 0.000,C 90.000,E1 129.725} C_DIS
LIN {X -0.035,Y -196.580,Z 1176.703,A 0.000,B 0.000,C 90.000,E1 126.457} C_DIS
LIN {X -0.042,Y -201.177,Z 1176.689,A 0.000,B 0.000,C 90.000,E1 124.119} C_DIS
LIN {X -0.101,Y -310.646,Z 1176.689,A 0.000,B 0.000,C 90.000,E1 124.119} C_DIS
LIN {X 0.078,Y -314.484,Z 1176.689,A 0.000,B 0.000,C 90.000,E1 123.992} C_DIS
LIN {X 0.077,Y -317.306,Z 1176.688,A 0.000,B 0.000,C 90.000,E1 123.833} C_DIS
LIN {X 0.016,Y -321.005,Z 1176.686,A 0.000,B 0.000,C 90.000,E1 123.499} C_DIS
LIN {X 0.080,Y -324.532,Z 1176.683,A 0.000,B 0.000,C 90.000,E1 122.959} C_DIS
LIN {X -0.108,Y -326.020,Z 1176.681,A 0.000,B 0.000,C 90.000,E1 122.673} C_DIS
LIN {X -0.025,Y -339.343,Z 1176.662,A 0.000,B 0.000,C 90.000,E1 119.205} C_DIS
LIN {X -0.004,Y -351.725,Z 1176.647,A 0.000,B 0.000,C 90.000,E1 116.437} C_DIS
LIN {X 0.071,Y -365.606,Z 1176.632,A 0.000,B 0.000,C 90.000,E1 113.718} C_DIS
LIN {X 0.138,Y -379.298,Z 1176.619,A 0.000,B 0.000,C 90.000,E1 111.354} C_DIS
LIN {X -0.098,Y -394.364,Z 1176.606,A 0.000,B 0.000,C 90.000,E1 109.087} C_DIS
LIN {X 0.156,Y -410.912,Z 1176.594,A 0.000,B 0.000,C 90.000,E1 106.804} C_DIS
LIN {X -0.097,Y -429.060,Z 1176.581,A 0.000,B 0.000,C 90.000,E1 104.647} C_DIS
LIN {X -0.084,Y -448.722,Z 1176.570,A 0.000,B 0.000,C 90.000,E1 102.535} C_DIS
LIN {X -0.187,Y -469.049,Z 1176.559,A 0.000,B 0.000,C 90.000,E1 100.602} C_DIS
LIN {X -0.145,Y -471.339,Z 1176.557,A 0.000,B 0.000,C 90.000,E1 100.366} C_DIS
LIN {X -0.186,Y -473.069,Z 1176.556,A 0.000,B 0.000,C 90.000,E1 100.141} C_DIS
LIN {X 0.141,Y -474.512,Z 1176.555,A 0.000,B 0.000,C 90.000,E1 99.849} C_DIS
LIN {X -0.001,Y -475.587,Z 1176.553,A 0.000,B 0.000,C 90.000,E1 99.613} C_DIS
LIN {X 0.124,Y -476.846,Z 1176.551,A 0.000,B 0.000,C 90.000,E1 99.095} C_DIS
LIN {X -0.142,Y -477.094,Z 1176.548,A 0.000,B 0.000,C 90.000,E1 98.624} C_DIS
LIN {X -0.001,Y -476.372,Z 1176.545,A 0.000,B 0.000,C 90.000,E1 98.106} C_DIS
LIN {X 0.142,Y -474.565,Z 1176.542,A 0.000,B 0.000,C 90.000,E1 97.587} C_DIS
LIN {X 0.006,Y -473.150,Z 1176.541,A 0.000,B 0.000,C 90.000,E1 97.352} C_DIS
LIN {X -0.066,Y -458.704,Z 1176.530,A 0.000,B 0.000,C 90.000,E1 95.334} C_DIS
LIN {X -0.124,Y -441.105,Z 1176.515,A 0.000,B 0.000,C 90.000,E1 92.751} C_DIS
LIN {X -0.134,Y -423.257,Z 1176.499,A 0.000,B 0.000,C 90.000,E1 89.828} C_DIS
LIN {X -0.025,Y -409.878,Z 1176.485,A 0.000,B 0.000,C 90.000,E1 87.364} C_DIS
LIN {X 0.062,Y -399.589,Z 1176.475,A 0.000,B 0.000,C 90.000,E1 85.412} C_DIS
LIN {X 0.008,Y -387.805,Z 1176.462,A 0.000,B 0.000,C 90.000,E1 83.166} C_DIS
LIN {X 0.135,Y -377.532,Z 1176.451,A 0.000,B 0.000,C 90.000,E1 81.141} C_DIS
LIN {X 0.111,Y -368.416,Z 1176.441,A 0.000,B 0.000,C 90.000,E1 79.398} C_DIS
LIN {X -0.008,Y -359.010,Z 1176.431,A 0.000,B 0.000,C 90.000,E1 77.645} C_DIS
LIN {X 0.124,Y -349.401,Z 1176.421,A 0.000,B 0.000,C 90.000,E1 75.825} C_DIS
LIN {X -0.174,Y -338.065,Z 1176.410,A 0.000,B 0.000,C 90.000,E1 73.740} C_DIS
LIN {X -0.004,Y -325.368,Z 1176.396,A 0.000,B 0.000,C 90.000,E1 71.221} C_DIS
LIN {X 0.089,Y -311.726,Z 1176.380,A 0.000,B 0.000,C 90.000,E1 68.337} C_DIS
LIN {X -0.066,Y -297.453,Z 1176.362,A 0.000,B 0.000,C 90.000,E1 65.101} C_DIS
LIN {X -0.121,Y -285.436,Z 1176.345,A 0.000,B 0.000,C 90.000,E1 62.103} C_DIS
LIN {X -0.033,Y -272.832,Z 1176.326,A 0.000,B 0.000,C 90.000,E1 58.663} C_DIS
LIN {X -0.098,Y -263.214,Z 1176.310,A 0.000,B 0.000,C 90.000,E1 55.881} C_DIS
LIN {X 0.092,Y -251.825,Z 1176.291,A 0.000,B 0.000,C 90.000,E1 52.271} C_DIS
LIN {X 0.014,Y -241.205,Z 1176.270,A 0.000,B 0.000,C 90.000,E1 48.647} C_DIS
LIN {X 0.061,Y -231.387,Z 1176.250,A 0.000,B 0.000,C 90.000,E1 44.919} C_DIS
LIN {X -0.019,Y -222.510,Z 1176.229,A 0.000,B 0.000,C 90.000,E1 41.148} C_DIS
LIN {X 0.003,Y -214.400,Z 1176.207,A 0.000,B 0.000,C 90.000,E1 37.282} C_DIS
LIN {X -0.054,Y -207.043,Z 1176.185,A 0.000,B 0.000,C 90.000,E1 33.372} C_DIS
LIN {X 0.031,Y -200.404,Z 1176.163,A 0.000,B 0.000,C 90.000,E1 29.361} C_DIS
LIN {X -0.035,Y -194.521,Z 1176.141,A 0.000,B 0.000,C 90.000,E1 25.335} C_DIS
LIN {X 0.006,Y -189.522,Z 1176.118,A 0.000,B 0.000,C 90.000,E1 21.227} C_DIS
LIN {X -0.022,Y -185.377,Z 1176.095,A 0.000,B 0.000,C 90.000,E1 17.094} C_DIS
LIN {X 0.084,Y -182.274,Z 1176.072,A 0.000,B 0.000,C 90.000,E1 12.883} C_DIS
LIN {X 0.034,Y -179.513,Z 1176.039,A 0.000,B 0.000,C 90.000,E1 7.004} C_DIS
LIN {X 0.074,Y -180.546,Z 1175.969,A 0.000,B 0.000,C 90.000,E1 354.432} C_DIS
LIN {X 0.010,Y -183.504,Z 1175.941,A 0.000,B 0.000,C 90.000,E1 349.398} C_DIS
LIN {X -0.031,Y -187.037,Z 1175.918,A 0.000,B 0.000,C 90.000,E1 345.227} C_DIS
LIN {X -0.081,Y -191.497,Z 1175.895,A 0.000,B 0.000,C 90.000,E1 341.094} C_DIS
LIN {X -0.035,Y -196.676,Z 1175.872,A 0.000,B 0.000,C 90.000,E1 336.975} C_DIS
LIN {X -0.007,Y -201.359,Z 1175.854,A 0.000,B 0.000,C 90.000,E1 333.717} C_DIS
LIN {X 0.127,Y -207.816,Z 1175.832,A 0.000,B 0.000,C 90.000,E1 329.665} C_DIS
LIN {X -0.042,Y -214.802,Z 1175.810,A 0.000,B 0.000,C 90.000,E1 325.754} C_DIS
LIN {X -0.068,Y -220.945,Z 1175.792,A 0.000,B 0.000,C 90.000,E1 322.637} C_DIS
LIN {X -0.016,Y -227.970,Z 1175.775,A 0.000,B 0.000,C 90.000,E1 319.542} C_DIS
LIN {X 0.019,Y -236.066,Z 1175.758,A 0.000,B 0.000,C 90.000,E1 316.500} C_DIS
LIN {X -0.067,Y -245.263,Z 1175.742,A 0.000,B 0.000,C 90.000,E1 313.542} C_DIS
LIN {X -0.074,Y -255.488,Z 1175.726,A 0.000,B 0.000,C 90.000,E1 310.620} C_DIS
LIN {X 0.118,Y -268.219,Z 1175.708,A 0.000,B 0.000,C 90.000,E1 307.363} C_DIS
LIN {X -0.021,Y -279.229,Z 1175.694,A 0.000,B 0.000,C 90.000,E1 304.945} C_DIS
LIN {X 0.026,Y -289.631,Z 1175.683,A 0.000,B 0.000,C 90.000,E1 302.880} C_DIS
LIN {X 0.022,Y -307.013,Z 1175.666,A 0.000,B 0.000,C 90.000,E1 299.873} C_DIS
LIN {X 0.148,Y -319.709,Z 1175.655,A 0.000,B 0.000,C 90.000,E1 297.897} C_DIS
LIN {X -0.180,Y -331.457,Z 1175.646,A 0.000,B 0.000,C 90.000,E1 296.360} C_DIS
LIN {X -0.161,Y -349.536,Z 1175.634,A 0.000,B 0.000,C 90.000,E1 294.207} C_DIS
LIN {X -0.087,Y -365.517,Z 1175.625,A 0.000,B 0.000,C 90.000,E1 292.461} C_DIS
LIN {X -0.046,Y -389.844,Z 1175.612,A 0.000,B 0.000,C 90.000,E1 290.120} C_DIS
LIN {X 0.205,Y -400.497,Z 1175.606,A 0.000,B 0.000,C 90.000,E1 289.087} C_DIS
LIN {X -0.087,Y -410.886,Z 1175.601,A 0.000,B 0.000,C 90.000,E1 288.127} C_DIS
LIN {X -0.129,Y -421.015,Z 1175.595,A 0.000,B 0.000,C 90.000,E1 287.094} C_DIS
LIN {X 0.123,Y -428.457,Z 1175.590,A 0.000,B 0.000,C 90.000,E1 286.260} C_DIS
LIN {X -0.075,Y -435.503,Z 1175.586,A 0.000,B 0.000,C 90.000,E1 285.481} C_DIS
LIN {X 0.085,Y -442.026,Z 1175.582,A 0.000,B 0.000,C 90.000,E1 284.662} C_DIS
LIN {X -0.017,Y -447.689,Z 1175.577,A 0.000,B 0.000,C 90.000,E1 283.883} C_DIS
LIN {X -0.176,Y -452.724,Z 1175.573,A 0.000,B 0.000,C 90.000,E1 283.119} C_DIS
LIN {X 0.149,Y -457.163,Z 1175.568,A 0.000,B 0.000,C 90.000,E1 282.299} C_DIS
LIN {X 0.074,Y -460.942,Z 1175.564,A 0.000,B 0.000,C 90.000,E1 281.535} C_DIS
LIN {X -0.063,Y -464.104,Z 1175.560,A 0.000,B 0.000,C 90.000,E1 280.782} C_DIS
LIN {X 0.073,Y -465.959,Z 1175.557,A 0.000,B 0.000,C 90.000,E1 280.254} C_DIS
LIN {X 0.213,Y -467.598,Z 1175.554,A 0.000,B 0.000,C 90.000,E1 279.726} C_DIS
LIN {X -0.177,Y -469.034,Z 1175.551,A 0.000,B 0.000,C 90.000,E1 279.265} C_DIS
LIN {X -0.093,Y -470.253,Z 1175.549,A 0.000,B 0.000,C 90.000,E1 278.746} C_DIS
LIN {X 0.070,Y -471.222,Z 1175.546,A 0.000,B 0.000,C 90.000,E1 278.219} C_DIS
LIN {X 0.173,Y -471.903,Z 1175.543,A 0.000,B 0.000,C 90.000,E1 277.701} C_DIS
LIN {X -0.186,Y -472.204,Z 1175.540,A 0.000,B 0.000,C 90.000,E1 277.239} C_DIS
LIN {X -0.072,Y -472.031,Z 1175.537,A 0.000,B 0.000,C 90.000,E1 276.720} C_DIS
LIN {X 0.044,Y -471.467,Z 1175.534,A 0.000,B 0.000,C 90.000,E1 276.201} C_DIS
LIN {X 0.158,Y -470.473,Z 1175.532,A 0.000,B 0.000,C 90.000,E1 275.682} C_DIS
LIN {X -0.199,Y -469.040,Z 1175.529,A 0.000,B 0.000,C 90.000,E1 275.220} C_DIS
LIN {X -0.096,Y -467.166,Z 1175.526,A 0.000,B 0.000,C 90.000,E1 274.702} C_DIS
LIN {X -0.038,Y -464.749,Z 1175.523,A 0.000,B 0.000,C 90.000,E1 274.188} C_DIS
LIN {X 0.037,Y -461.714,Z 1175.520,A 0.000,B 0.000,C 90.000,E1 273.669} C_DIS
LIN {X 0.068,Y -457.836,Z 1175.518,A 0.000,B 0.000,C 90.000,E1 273.154} C_DIS
LIN {X -0.130,Y -455.513,Z 1175.516,A 0.000,B 0.000,C 90.000,E1 272.922} C_DIS
LIN {X -0.026,Y -450.105,Z 1175.513,A 0.000,B 0.000,C 90.000,E1 272.407} C_DIS
LIN {X -0.152,Y -446.908,Z 1175.512,A 0.000,B 0.000,C 90.000,E1 272.178} C_DIS
LIN {X 0.152,Y -440.328,Z 1175.510,A 0.000,B 0.000,C 90.000,E1 271.718} C_DIS
LIN {X 0.101,Y -433.399,Z 1175.508,A 0.000,B 0.000,C 90.000,E1 271.375} C_DIS
LIN {X 0.104,Y -426.529,Z 1175.506,A 0.000,B 0.000,C 90.000,E1 271.088} C_DIS
LIN {X -0.011,Y -419.474,Z 1175.505,A 0.000,B 0.000,C 90.000,E1 270.859} C_DIS
LIN {X 0.129,Y -412.218,Z 1175.504,A 0.000,B 0.000,C 90.000,E1 270.630} C_DIS
LIN {X 0.000,Y -401.570,Z 1175.502,A 0.000,B 0.000,C 90.000,E1 270.401} C_DIS
LIN {X 0.175,Y -390.731,Z 1175.501,A 0.000,B 0.000,C 90.000,E1 270.172} C_DIS
LIN {X 0.159,Y -382.981,Z 1175.500,A 0.000,B 0.000,C 90.000,E1 270.057} C_DIS
LIN {X 0.047,Y -374.786,Z 1175.500,A 0.000,B 0.000,C 90.000,E1 270.000} C_DIS
LIN {X -0.160,Y -366.498,Z 1175.500,A 0.000,B 0.000,C 90.000,E1 270.000} C_DIS
LIN {X 0.078,Y -181.555,Z 1175.500,A 0.000,B 0.000,C 90.000,E1 269.943} C_DIS
LIN {X -0.081,Y -180.827,Z 1175.471,A 0.000,B 0.000,C 90.000,E1 264.894} C_DIS
LIN {X -0.002,Y -178.932,Z 1175.443,A 0.000,B 0.000,C 90.000,E1 259.803} C_DIS
LIN {X 0.037,Y -175.980,Z 1175.415,A 0.000,B 0.000,C 90.000,E1 254.700} C_DIS
LIN {X -0.018,Y -175.471,Z 1175.410,A 0.000,B 0.000,C 90.000,E1 253.866} C_DIS
LIN {X 0.038,Y -172.220,Z 1175.387,A 0.000,B 0.000,C 90.000,E1 249.571} C_DIS
LIN {X 0.016,Y -171.696,Z 1175.382,A 0.000,B 0.000,C 90.000,E1 248.720} C_DIS
LIN {X 0.091,Y -167.290,Z 1175.353,A 0.000,B 0.000,C 90.000,E1 243.512} C_DIS
LIN {X 0.025,Y -166.667,Z 1175.348,A 0.000,B 0.000,C 90.000,E1 242.666} C_DIS
LIN {X -0.061,Y -162.650,Z 1175.324,A 0.000,B 0.000,C 90.000,E1 238.329} C_DIS
LIN {X 0.002,Y -161.338,Z 1175.314,A 0.000,B 0.000,C 90.000,E1 236.548} C_DIS
LIN {X 0.044,Y -157.333,Z 1175.290,A 0.000,B 0.000,C 90.000,E1 232.110} C_DIS
LIN {X -0.023,Y -155.317,Z 1175.275,A 0.000,B 0.000,C 90.000,E1 229.461} C_DIS
LIN {X 0.015,Y -151.672,Z 1175.250,A 0.000,B 0.000,C 90.000,E1 224.960} C_DIS
LIN {X -0.044,Y -150.537,Z 1175.240,A 0.000,B 0.000,C 90.000,E1 223.176} C_DIS
LIN {X -0.010,Y -147.262,Z 1175.215,A 0.000,B 0.000,C 90.000,E1 218.624} C_DIS
LIN {X 0.046,Y -145.289,Z 1175.194,A 0.000,B 0.000,C 90.000,E1 214.945} C_DIS
LIN {X -0.045,Y -142.388,Z 1175.164,A 0.000,B 0.000,C 90.000,E1 209.461} C_DIS
LIN {X 0.002,Y -141.367,Z 1175.148,A 0.000,B 0.000,C 90.000,E1 206.668} C_DIS
LIN {X -0.020,Y -139.344,Z 1175.112,A 0.000,B 0.000,C 90.000,E1 200.174} C_DIS
LIN {X -0.015,Y -139.015,Z 1175.102,A 0.000,B 0.000,C 90.000,E1 198.308} C_DIS
LIN {X -0.019,Y -138.342,Z 1175.055,A 0.000,B 0.000,C 90.000,E1 189.905} C_DIS
LIN {X 0.001,Y -139.395,Z 1175.008,A 0.000,B 0.000,C 90.000,E1 181.489} C_DIS
LIN {X 0.054,Y -141.297,Z 1174.972,A 0.000,B 0.000,C 90.000,E1 174.951} C_DIS
LIN {X 0.012,Y -142.659,Z 1174.957,A 0.000,B 0.000,C 90.000,E1 172.186} C_DIS
LIN {X -0.038,Y -145.002,Z 1174.931,A 0.000,B 0.000,C 90.000,E1 167.589} C_DIS
LIN {X -0.049,Y -147.629,Z 1174.911,A 0.000,B 0.000,C 90.000,E1 163.921} C_DIS
LIN {X 0.029,Y -150.257,Z 1174.890,A 0.000,B 0.000,C 90.000,E1 160.242} C_DIS
LIN {X 0.043,Y -153.655,Z 1174.870,A 0.000,B 0.000,C 90.000,E1 156.613} C_DIS
LIN {X -0.040,Y -157.070,Z 1174.850,A 0.000,B 0.000,C 90.000,E1 153.050} C_DIS
LIN {X 0.039,Y -161.203,Z 1174.830,A 0.000,B 0.000,C 90.000,E1 149.459} C_DIS
LIN {X -0.013,Y -163.294,Z 1174.821,A 0.000,B 0.000,C 90.000,E1 147.709} C_DIS
LIN {X -0.003,Y -167.740,Z 1174.801,A 0.000,B 0.000,C 90.000,E1 144.196} C_DIS
LIN {X -0.091,Y -171.558,Z 1174.787,A 0.000,B 0.000,C 90.000,E1 141.618} C_DIS
